LIN {X 0,Y 229.737,Z 261.729,A -85,B 0,C 180,E1 -19927.308,E2 -19927.308} C_VEL
LIN {X 0,Y 228.307,Z 255.768,A -85,B 0,C 180,E1 -19931.044,E2 -19931.044} C_VEL
LIN {X 0,Y 227.847,Z 253.604,A -85,B 0,C 180,E1 -19932.574,E2 -19932.574} C_VEL
LIN {X 0,Y 227.809,Z 253.608,A -85,B 0,C 180,E1 -19937.256,E2 -19937.256} C_VEL
LIN {X 0,Y 227.847,Z 253.599,A -85,B 0,C 180,E1 -19941.908,E2 -19941.908} C_VEL
LIN {X 0,Y 227.882,Z 253.572,A -85,B 0,C 180,E1 -19946.376,E2 -19946.376} C_VEL
LIN {X 0,Y 227.906,Z 253.589,A -85,B 0,C 180,E1 -19950.435,E2 -19950.435} C_VEL
LIN {X 0,Y 227.93,Z 253.565,A -85,B 0,C 180,E1 -19954.425,E2 -19954.425} C_VEL
LIN {X 0,Y 227.963,Z 253.579,A -85,B 0,C 180,E1 -19958.286,E2 -19958.286} C_VEL
LIN {X 0,Y 228.005,Z 253.549,A -85,B 0,C 180,E1 -19962.85,E2 -19962.85} C_VEL
LIN {X 0,Y 228.067,Z 253.561,A -85,B 0,C 180,E1 -19967.542,E2 -19967.542} C_VEL
LIN {X 0,Y 228.255,Z 253.506,A -85,B 0,C 180,E1 -19971.143,E2 -19971.143} C_VEL
LIN {X 0,Y 228.306,Z 253.525,A -85,B 0,C 180,E1 -19972.926,E2 -19972.926} C_VEL
LIN {X 0,Y 228.553,Z 253.484,A -85,B 0,C 180,E1 -19978.237,E2 -19978.237} C_VEL
LIN {X 0,Y 228.554,Z 253.477,A -85,B 0,C 180,E1 -19981.761,E2 -19981.761} C_VEL
LIN {X 0,Y 228.339,Z 253.528,A -85,B 0,C 180,E1 -19987.071,E2 -19987.071} C_VEL
LIN {X 0,Y 228.145,Z 253.521,A -85,B 0,C 180,E1 -19990.65,E2 -19990.65} C_VEL
LIN {X 0,Y 228.064,Z 253.576,A -85,B 0,C 180,E1 -19994.271,E2 -19994.271} C_VEL
LIN {X 0,Y 228.001,Z 253.548,A -85,B 0,C 180,E1 -19997.952,E2 -19997.952} C_VEL
LIN {X 0,Y 227.915,Z 253.589,A -85,B 0,C 180,E1 -20002.32,E2 -20002.32} C_VEL
LIN {X 0,Y 227.939,Z 253.559,A -85,B 0,C 180,E1 -20006.601,E2 -20006.601} C_VEL
LIN {X 0,Y 227.895,Z 253.595,A -85,B 0,C 180,E1 -20010.29,E2 -20010.29} C_VEL
LIN {X 0,Y 227.887,Z 253.575,A -85,B 0,C 180,E1 -20013.717,E2 -20013.717} C_VEL
LIN {X 0,Y 227.869,Z 253.602,A -85,B 0,C 180,E1 -20018.085,E2 -20018.085} C_VEL
LIN {X 0,Y 227.907,Z 253.592,A -85,B 0,C 180,E1 -20022.719,E2 -20022.719} C_VEL
LIN {X 0,Y 227.818,Z 253.543,A -85,B 0,C 180,E1 -20027.259,E2 -20027.259} C_VEL
LIN {X 0,Y 227.867,Z 253.603,A -85,B 0,C 180,E1 -20031.914,E2 -20031.914} C_VEL
LIN {X 0,Y 227.936,Z 253.841,A -85,B 0,C 180,E1 -20032.886,E2 -20032.886} C_VEL
LIN {X 0,Y 228.192,Z 254.913,A -85,B 0,C 180,E1 -20033.201,E2 -20033.201} C_VEL
LIN {X 0,Y 229.812,Z 257.623,A -85,B 0,C 180,E1 -20033.627,E2 -20033.627} C_VEL
LIN {X 0,Y 237.856,Z 271.226,A -85,B 0,C 180,E1 -20035.542,E2 -20035.542} C_VEL
LIN {X 0,Y 245.107,Z 285.042,A -85,B 0,C 180,E1 -20037.18,E2 -20037.18} C_VEL
LIN {X 0,Y 252.288,Z 298.523,A -85,B 0,C 180,E1 -20038.675,E2 -20038.675} C_VEL
LIN {X 0,Y 261.001,Z 311.411,A -85,B 0,C 180,E1 -20040.242,E2 -20040.242} C_VEL
LIN {X 0,Y 271.599,Z 324.085,A -85,B 0,C 180,E1 -20041.896,E2 -20041.896} C_VEL
LIN {X 0,Y 286.219,Z 338.842,A -85,B 0,C 180,E1 -20043.865,E2 -20043.865} C_VEL
LIN {X 0,Y 299.817,Z 350.422,A -85,B 0,C 180,E1 -20045.476,E2 -20045.476} C_VEL
LIN {X 0,Y 307.35,Z 356.574,A -85,B 0,C 180,E1 -20046.45,E2 -20046.45} C_VEL
LIN {X 0,Y 315.79,Z 363.116,A -85,B 0,C 180,E1 -20047.769,E2 -20047.769} C_VEL
LIN {X 0,Y 323.958,Z 369.179,A -85,B 0,C 180,E1 -20049.245,E2 -20049.245} C_VEL
LIN {X 0,Y 332.274,Z 375.418,A -85,B 0,C 180,E1 -20050.97,E2 -20050.97} C_VEL
LIN {X 0,Y 339.722,Z 380.424,A -85,B 0,C 180,E1 -20052.688,E2 -20052.688} C_VEL
LIN {X 0,Y 346.418,Z 385.336,A -85,B 0,C 180,E1 -20054.487,E2 -20054.487} C_VEL
LIN {X 0,Y 351.921,Z 388.859,A -85,B 0,C 180,E1 -20056.134,E2 -20056.134} C_VEL
LIN {X 0,Y 355.938,Z 391.12,A -85,B 0,C 180,E1 -20057.456,E2 -20057.456} C_VEL
LIN {X 0,Y 359.128,Z 393.588,A -85,B 0,C 180,E1 -20058.715,E2 -20058.715} C_VEL
LIN {X 0,Y 363.313,Z 396.472,A -85,B 0,C 180,E1 -20060.589,E2 -20060.589} C_VEL
LIN {X 0,Y 366.571,Z 398.29,A -85,B 0,C 180,E1 -20062.287,E2 -20062.287} C_VEL
LIN {X 0,Y 368.408,Z 399.219,A -85,B 0,C 180,E1 -20063.428,E2 -20063.428} C_VEL
LIN {X 0,Y 369.965,Z 399.891,A -85,B 0,C 180,E1 -20064.55,E2 -20064.55} C_VEL
LIN {X 0,Y 371.247,Z 400.329,A -85,B 0,C 180,E1 -20065.657,E2 -20065.657} C_VEL
LIN {X 0,Y 372.236,Z 400.623,A -85,B 0,C 180,E1 -20066.753,E2 -20066.753} C_VEL
LIN {X 0,Y 372.866,Z 401.006,A -85,B 0,C 180,E1 -20067.84,E2 -20067.84} C_VEL
LIN {X 0,Y 373.231,Z 401.261,A -85,B 0,C 180,E1 -20068.921,E2 -20068.921} C_VEL
LIN {X 0,Y 373.406,Z 401.192,A -85,B 0,C 180,E1 -20070,E2 -20070} C_VEL
LIN {X 0,Y 373.242,Z 401.224,A -85,B 0,C 180,E1 -20071.079,E2 -20071.079} C_VEL
LIN {X 0,Y 372.799,Z 400.889,A -85,B 0,C 180,E1 -20072.374,E2 -20072.374} C_VEL
LIN {X 0,Y 371.247,Z 400.335,A -85,B 0,C 180,E1 -20074.343,E2 -20074.343} C_VEL
LIN {X 0,Y 369.963,Z 399.917,A -85,B 0,C 180,E1 -20075.45,E2 -20075.45} C_VEL
LIN {X 0,Y 368.056,Z 399.053,A -85,B 0,C 180,E1 -20076.821,E2 -20076.821} C_VEL
LIN {X 0,Y 364.414,Z 397.149,A -85,B 0,C 180,E1 -20078.875,E2 -20078.875} C_VEL
LIN {X 0,Y 361.943,Z 395.593,A -85,B 0,C 180,E1 -20080.064,E2 -20080.064} C_VEL
LIN {X 0,Y 357.635,Z 392.463,A -85,B 0,C 180,E1 -20081.885,E2 -20081.885} C_VEL
LIN {X 0,Y 355.91,Z 391.059,A -85,B 0,C 180,E1 -20082.545,E2 -20082.545} C_VEL
LIN {X 0,Y 351.917,Z 388.848,A -85,B 0,C 180,E1 -20083.866,E2 -20083.866} C_VEL
LIN {X 0,Y 345.895,Z 385.025,A -85,B 0,C 180,E1 -20085.654,E2 -20085.654} C_VEL
LIN {X 0,Y 339.248,Z 380.069,A -85,B 0,C 180,E1 -20087.431,E2 -20087.431} C_VEL
LIN {X 0,Y 331.554,Z 374.906,A -85,B 0,C 180,E1 -20089.184,E2 -20089.184} C_VEL
LIN {X 0,Y 323.397,Z 368.785,A -85,B 0,C 180,E1 -20090.86,E2 -20090.86} C_VEL
LIN {X 0,Y 315.566,Z 362.953,A -85,B 0,C 180,E1 -20092.266,E2 -20092.266} C_VEL
LIN {X 0,Y 307.371,Z 356.596,A -85,B 0,C 180,E1 -20093.548,E2 -20093.548} C_VEL
LIN {X 0,Y 299.818,Z 350.408,A -85,B 0,C 180,E1 -20094.525,E2 -20094.525} C_VEL
LIN {X 0,Y 286.642,Z 339.218,A -85,B 0,C 180,E1 -20096.082,E2 -20096.082} C_VEL
LIN {X 0,Y 271.943,Z 324.45,A -85,B 0,C 180,E1 -20098.055,E2 -20098.055} C_VEL
LIN {X 0,Y 261.435,Z 311.99,A -85,B 0,C 180,E1 -20099.685,E2 -20099.685} C_VEL
LIN {X 0,Y 252.682,Z 299.196,A -85,B 0,C 180,E1 -20101.248,E2 -20101.248} C_VEL
LIN {X 0,Y 245.461,Z 285.814,A -85,B 0,C 180,E1 -20102.74,E2 -20102.74} C_VEL
LIN {X 0,Y 239.261,Z 273.837,A -85,B 0,C 180,E1 -20104.133,E2 -20104.133} C_VEL
LIN {X 0,Y 231.483,Z 260.425,A -85,B 0,C 180,E1 -20105.961,E2 -20105.961} C_VEL
LIN {X 0,Y 229.703,Z 257.505,A -85,B 0,C 180,E1 -20106.397,E2 -20106.397} C_VEL
LIN {X 0,Y 228.093,Z 254.532,A -85,B 0,C 180,E1 -20106.86,E2 -20106.86} C_VEL
LIN {X 0,Y 227.902,Z 253.655,A -85,B 0,C 180,E1 -20107.312,E2 -20107.312} C_VEL
LIN {X 0,Y 227.832,Z 253.551,A -85,B 0,C 180,E1 -20110.375,E2 -20110.375} C_VEL
LIN {X 0,Y 227.854,Z 253.579,A -85,B 0,C 180,E1 -20115.187,E2 -20115.187} C_VEL
LIN {X 0,Y 227.907,Z 253.585,A -85,B 0,C 180,E1 -20117.739,E2 -20117.739} C_VEL
LIN {X 0,Y 227.869,Z 253.602,A -85,B 0,C 180,E1 -20121.915,E2 -20121.915} C_VEL
LIN {X 0,Y 227.888,Z 253.575,A -85,B 0,C 180,E1 -20126.374,E2 -20126.374} C_VEL
LIN {X 0,Y 227.902,Z 253.583,A -85,B 0,C 180,E1 -20130.437,E2 -20130.437} C_VEL
LIN {X 0,Y 227.923,Z 253.572,A -85,B 0,C 180,E1 -20134.426,E2 -20134.426} C_VEL
LIN {X 0,Y 227.946,Z 253.577,A -85,B 0,C 180,E1 -20138.287,E2 -20138.287} C_VEL
LIN {X 0,Y 228.033,Z 253.555,A -85,B 0,C 180,E1 -20142.827,E2 -20142.827} C_VEL
LIN {X 0,Y 228.072,Z 253.556,A -85,B 0,C 180,E1 -20147.544,E2 -20147.544} C_VEL
LIN {X 0,Y 228.267,Z 253.509,A -85,B 0,C 180,E1 -20151.146,E2 -20151.146} C_VEL
LIN {X 0,Y 228.339,Z 253.528,A -85,B 0,C 180,E1 -20152.929,E2 -20152.929} C_VEL
LIN {X 0,Y 228.554,Z 253.477,A -85,B 0,C 180,E1 -20158.239,E2 -20158.239} C_VEL
LIN {X 0,Y 228.553,Z 253.484,A -85,B 0,C 180,E1 -20161.763,E2 -20161.763} C_VEL
LIN {X 0,Y 228.306,Z 253.525,A -85,B 0,C 180,E1 -20167.074,E2 -20167.074} C_VEL
LIN {X 0,Y 228.145,Z 253.523,A -85,B 0,C 180,E1 -20170.652,E2 -20170.652} C_VEL
LIN {X 0,Y 228.046,Z 253.575,A -85,B 0,C 180,E1 -20174.274,E2 -20174.274} C_VEL
LIN {X 0,Y 227.971,Z 253.546,A -85,B 0,C 180,E1 -20177.957,E2 -20177.957} C_VEL
LIN {X 0,Y 227.931,Z 253.589,A -85,B 0,C 180,E1 -20182.33,E2 -20182.33} C_VEL
LIN {X 0,Y 227.943,Z 253.556,A -85,B 0,C 180,E1 -20186.603,E2 -20186.603} C_VEL
LIN {X 0,Y 227.898,Z 253.596,A -85,B 0,C 180,E1 -20190.292,E2 -20190.292} C_VEL
LIN {X 0,Y 227.88,Z 253.572,A -85,B 0,C 180,E1 -20193.721,E2 -20193.721} C_VEL
LIN {X 0,Y 227.847,Z 253.599,A -85,B 0,C 180,E1 -20198.092,E2 -20198.092} C_VEL
LIN {X 0,Y 227.809,Z 253.608,A -85,B 0,C 180,E1 -20202.744,E2 -20202.744} C_VEL
LIN {X 0,Y 227.847,Z 253.614,A -85,B 0,C 180,E1 -20207.426,E2 -20207.426} C_VEL
LIN {X 0,Y 229.235,Z 259.354,A -85,B 0,C 180,E1 -20211.232,E2 -20211.232} C_VEL
LIN {X 0,Y 230.078,Z 263.105,A -85,B 0,C 180,E1 -20213.398,E2 -20213.398} C_VEL
LIN {X 0,Y 231.753,Z 266.915,A -85,B 0,C 180,E1 -20213.949,E2 -20213.949} C_VEL
LIN {X 0,Y 238.319,Z 280.506,A -85,B 0,C 180,E1 -20215.569,E2 -20215.569} C_VEL
LIN {X 0,Y 243.678,Z 293.124,A -85,B 0,C 180,E1 -20216.858,E2 -20216.858} C_VEL
LIN {X 0,Y 247.512,Z 314.657,A -85,B 0,C 180,E1 -20218.153,E2 -20218.153} C_VEL
LIN {X 0,Y 248.126,Z 318.744,A -85,B 0,C 180,E1 -20218.376,E2 -20218.376} C_VEL
LIN {X 0,Y 248.041,Z 322.266,A -85,B 0,C 180,E1 -20218.481,E2 -20218.481} C_VEL
LIN {X 0,Y 247.222,Z 328.114,A -85,B 0,C 180,E1 -20218.56,E2 -20218.56} C_VEL
LIN {X 0,Y 241.565,Z 347.124,A -85,B 0,C 180,E1 -20218.394,E2 -20218.394} C_VEL
LIN {X 0,Y 240.803,Z 352.968,A -85,B 0,C 180,E1 -20218.483,E2 -20218.483} C_VEL
LIN {X 0,Y 239.893,Z 372.687,A -85,B 0,C 180,E1 -20219.125,E2 -20219.125} C_VEL
LIN {X 0,Y 238.345,Z 386.631,A -85,B 0,C 180,E1 -20219.916,E2 -20219.916} C_VEL
LIN {X 0,Y 236.753,Z 397.271,A -85,B 0,C 180,E1 -20220.795,E2 -20220.795} C_VEL
LIN {X 0,Y 235.174,Z 405.775,A -85,B 0,C 180,E1 -20221.679,E2 -20221.679} C_VEL
LIN {X 0,Y 233.292,Z 415.049,A -85,B 0,C 180,E1 -20222.894,E2 -20222.894} C_VEL
LIN {X 0,Y 231.234,Z 423.992,A -85,B 0,C 180,E1 -20224.335,E2 -20224.335} C_VEL
LIN {X 0,Y 228.992,Z 432.516,A -85,B 0,C 180,E1 -20226.005,E2 -20226.005} C_VEL
LIN {X 0,Y 227.037,Z 439.733,A -85,B 0,C 180,E1 -20227.716,E2 -20227.716} C_VEL
LIN {X 0,Y 225.477,Z 445.825,A -85,B 0,C 180,E1 -20229.433,E2 -20229.433} C_VEL
LIN {X 0,Y 223.485,Z 452.473,A -85,B 0,C 180,E1 -20231.671,E2 -20231.671} C_VEL
LIN {X 0,Y 222.243,Z 456.976,A -85,B 0,C 180,E1 -20233.465,E2 -20233.465} C_VEL
LIN {X 0,Y 220.61,Z 462.466,A -85,B 0,C 180,E1 -20236.177,E2 -20236.177} C_VEL
LIN {X 0,Y 219.587,Z 466.796,A -85,B 0,C 180,E1 -20238.929,E2 -20238.929} C_VEL
LIN {X 0,Y 219.086,Z 469.166,A -85,B 0,C 180,E1 -20240.77,E2 -20240.77} C_VEL
LIN {X 0,Y 218.737,Z 470.968,A -85,B 0,C 180,E1 -20242.616,E2 -20242.616} C_VEL
LIN {X 0,Y 218.501,Z 473.423,A -85,B 0,C 180,E1 -20246.312,E2 -20246.312} C_VEL
LIN {X 0,Y 218.524,Z 474.016,A -85,B 0,C 180,E1 -20248.157,E2 -20248.157} C_VEL
LIN {X 0,Y 218.623,Z 474.174,A -85,B 0,C 180,E1 -20250,E2 -20250} C_VEL
LIN {X 0,Y 218.524,Z 474.016,A -85,B 0,C 180,E1 -20251.843,E2 -20251.843} C_VEL
LIN {X 0,Y 218.484,Z 473.159,A -85,B 0,C 180,E1 -20254.292,E2 -20254.292} C_VEL
LIN {X 0,Y 218.705,Z 470.967,A -85,B 0,C 180,E1 -20257.385,E2 -20257.385} C_VEL
LIN {X 0,Y 219.314,Z 468.015,A -85,B 0,C 180,E1 -20260.151,E2 -20260.151} C_VEL
LIN {X 0,Y 220.223,Z 464.022,A -85,B 0,C 180,E1 -20262.908,E2 -20262.908} C_VEL
LIN {X 0,Y 221.649,Z 458.891,A -85,B 0,C 180,E1 -20265.635,E2 -20265.635} C_VEL
LIN {X 0,Y 223.148,Z 453.628,A -85,B 0,C 180,E1 -20267.883,E2 -20267.883} C_VEL
LIN {X 0,Y 225.05,Z 447.314,A -85,B 0,C 180,E1 -20270.091,E2 -20270.091} C_VEL
LIN {X 0,Y 226.622,Z 441.361,A -85,B 0,C 180,E1 -20271.848,E2 -20271.848} C_VEL
LIN {X 0,Y 228.482,Z 434.435,A -85,B 0,C 180,E1 -20273.57,E2 -20273.57} C_VEL
LIN {X 0,Y 230.686,Z 426.261,A -85,B 0,C 180,E1 -20275.247,E2 -20275.247} C_VEL
LIN {X 0,Y 232.7,Z 417.752,A -85,B 0,C 180,E1 -20276.696,E2 -20276.696} C_VEL
LIN {X 0,Y 234.562,Z 409.039,A -85,B 0,C 180,E1 -20277.915,E2 -20277.915} C_VEL
LIN {X 0,Y 236.239,Z 400.291,A -85,B 0,C 180,E1 -20278.91,E2 -20278.91} C_VEL
LIN {X 0,Y 237.837,Z 390.494,A -85,B 0,C 180,E1 -20279.789,E2 -20279.789} C_VEL
LIN {X 0,Y 239.069,Z 380.72,A -85,B 0,C 180,E1 -20280.46,E2 -20280.46} C_VEL
LIN {X 0,Y 240.014,Z 370.366,A -85,B 0,C 180,E1 -20280.964,E2 -20280.964} C_VEL
LIN {X 0,Y 241.204,Z 343.742,A -85,B 0,C 180,E1 -20281.774,E2 -20281.774} C_VEL
LIN {X 0,Y 241.982,Z 319.229,A -85,B 0,C 180,E1 -20282.501,E2 -20282.501} C_VEL
LIN {X 0,Y 238.66,Z 299.408,A -85,B 0,C 180,E1 -20283.704,E2 -20283.704} C_VEL
LIN {X 0,Y 237.524,Z 294.652,A -85,B 0,C 180,E1 -20284.056,E2 -20284.056} C_VEL
LIN {X 0,Y 230.872,Z 279.383,A -85,B 0,C 180,E1 -20285.74,E2 -20285.74} C_VEL
LIN {X 0,Y 224.408,Z 266.483,A -85,B 0,C 180,E1 -20287.435,E2 -20287.435} C_VEL
LIN {X 0,Y 222.795,Z 262.883,A -85,B 0,C 180,E1 -20287.999,E2 -20287.999} C_VEL
LIN {X 0,Y 221.307,Z 256.828,A -85,B 0,C 180,E1 -20291.827,E2 -20291.827} C_VEL
LIN {X 0,Y 220.77,Z 254.494,A -85,B 0,C 180,E1 -20293.614,E2 -20293.614} C_VEL
LIN {X 0,Y 220.769,Z 254.482,A -85,B 0,C 180,E1 -20298.046,E2 -20298.046} C_VEL
LIN {X 0,Y 220.826,Z 254.479,A -85,B 0,C 180,E1 -20302.792,E2 -20302.792} C_VEL
LIN {X 0,Y 220.818,Z 254.458,A -85,B 0,C 180,E1 -20307.243,E2 -20307.243} C_VEL
LIN {X 0,Y 220.828,Z 254.453,A -85,B 0,C 180,E1 -20311.484,E2 -20311.484} C_VEL
LIN {X 0,Y 220.869,Z 254.459,A -85,B 0,C 180,E1 -20315.564,E2 -20315.564} C_VEL
LIN {X 0,Y 220.889,Z 254.44,A -85,B 0,C 180,E1 -20319.513,E2 -20319.513} C_VEL
LIN {X 0,Y 220.987,Z 254.43,A -85,B 0,C 180,E1 -20323.367,E2 -20323.367} C_VEL
LIN {X 0,Y 221.004,Z 254.445,A -85,B 0,C 180,E1 -20327.137,E2 -20327.137} C_VEL
LIN {X 0,Y 221.195,Z 254.383,A -85,B 0,C 180,E1 -20330.858,E2 -20330.858} C_VEL
LIN {X 0,Y 221.129,Z 254.437,A -85,B 0,C 180,E1 -20334.528,E2 -20334.528} C_VEL
LIN {X 0,Y 221.511,Z 254.361,A -85,B 0,C 180,E1 -20338.181,E2 -20338.181} C_VEL
LIN {X 0,Y 221.512,Z 254.353,A -85,B 0,C 180,E1 -20341.817,E2 -20341.817} C_VEL
LIN {X 0,Y 221.271,Z 254.402,A -85,B 0,C 180,E1 -20347.298,E2 -20347.298} C_VEL
LIN {X 0,Y 221.067,Z 254.405,A -85,B 0,C 180,E1 -20350.995,E2 -20350.995} C_VEL
LIN {X 0,Y 220.996,Z 254.458,A -85,B 0,C 180,E1 -20354.738,E2 -20354.738} C_VEL
LIN {X 0,Y 220.919,Z 254.425,A -85,B 0,C 180,E1 -20358.549,E2 -20358.549} C_VEL
LIN {X 0,Y 220.883,Z 254.468,A -85,B 0,C 180,E1 -20362.675,E2 -20362.675} C_VEL
LIN {X 0,Y 220.881,Z 254.436,A -85,B 0,C 180,E1 -20367.013,E2 -20367.013} C_VEL
LIN {X 0,Y 220.836,Z 254.479,A -85,B 0,C 180,E1 -20370.767,E2 -20370.767} C_VEL
LIN {X 0,Y 220.813,Z 254.453,A -85,B 0,C 180,E1 -20374.951,E2 -20374.951} C_VEL
LIN {X 0,Y 220.853,Z 254.458,A -85,B 0,C 180,E1 -20379.525,E2 -20379.525} C_VEL
LIN {X 0,Y 220.864,Z 254.472,A -85,B 0,C 180,E1 -20382.957,E2 -20382.957} C_VEL
LIN {X 0,Y 220.776,Z 254.417,A -85,B 0,C 180,E1 -20388.049,E2 -20388.049} C_VEL
LIN {X 0,Y 220.836,Z 254.701,A -85,B 0,C 180,E1 -20391.491,E2 -20391.491} C_VEL
LIN {X 0,Y 221.128,Z 255.823,A -85,B 0,C 180,E1 -20391.848,E2 -20391.848} C_VEL
LIN {X 0,Y 222.822,Z 258.61,A -85,B 0,C 180,E1 -20392.322,E2 -20392.322} C_VEL
LIN {X 0,Y 228.235,Z 267.33,A -85,B 0,C 180,E1 -20393.706,E2 -20393.706} C_VEL
LIN {X 0,Y 237.078,Z 283.229,A -85,B 0,C 180,E1 -20395.845,E2 -20395.845} C_VEL
LIN {X 0,Y 246.332,Z 301.326,A -85,B 0,C 180,E1 -20397.916,E2 -20397.916} C_VEL
LIN {X 0,Y 254.709,Z 314.108,A -85,B 0,C 180,E1 -20399.51,E2 -20399.51} C_VEL
LIN {X 0,Y 263.082,Z 324.749,A -85,B 0,C 180,E1 -20400.913,E2 -20400.913} C_VEL
LIN {X 0,Y 275.601,Z 338.122,A -85,B 0,C 180,E1 -20402.747,E2 -20402.747} C_VEL
LIN {X 0,Y 285.746,Z 347.624,A -85,B 0,C 180,E1 -20404.06,E2 -20404.06} C_VEL
LIN {X 0,Y 296.508,Z 356.709,A -85,B 0,C 180,E1 -20405.344,E2 -20405.344} C_VEL
LIN {X 0,Y 304.924,Z 363.572,A -85,B 0,C 180,E1 -20406.474,E2 -20406.474} C_VEL
LIN {X 0,Y 312.969,Z 369.81,A -85,B 0,C 180,E1 -20407.749,E2 -20407.749} C_VEL
LIN {X 0,Y 321.3,Z 375.892,A -85,B 0,C 180,E1 -20409.254,E2 -20409.254} C_VEL
LIN {X 0,Y 329.279,Z 381.914,A -85,B 0,C 180,E1 -20410.917,E2 -20410.917} C_VEL
LIN {X 0,Y 335.925,Z 386.279,A -85,B 0,C 180,E1 -20412.433,E2 -20412.433} C_VEL
LIN {X 0,Y 343.054,Z 391.525,A -85,B 0,C 180,E1 -20414.334,E2 -20414.334} C_VEL
LIN {X 0,Y 348.695,Z 395.135,A -85,B 0,C 180,E1 -20416.004,E2 -20416.004} C_VEL
LIN {X 0,Y 352.899,Z 397.518,A -85,B 0,C 180,E1 -20417.376,E2 -20417.376} C_VEL
LIN {X 0,Y 357.622,Z 401.061,A -85,B 0,C 180,E1 -20419.292,E2 -20419.292} C_VEL
LIN {X 0,Y 361.371,Z 403.495,A -85,B 0,C 180,E1 -20421.049,E2 -20421.049} C_VEL
LIN {X 0,Y 363.553,Z 404.71,A -85,B 0,C 180,E1 -20422.223,E2 -20422.223} C_VEL
LIN {X 0,Y 365.44,Z 405.641,A -85,B 0,C 180,E1 -20423.374,E2 -20423.374} C_VEL
LIN {X 0,Y 367.1,Z 406.372,A -85,B 0,C 180,E1 -20424.567,E2 -20424.567} C_VEL
LIN {X 0,Y 368.316,Z 406.802,A -85,B 0,C 180,E1 -20425.623,E2 -20425.623} C_VEL
LIN {X 0,Y 369.338,Z 407.082,A -85,B 0,C 180,E1 -20426.727,E2 -20426.727} C_VEL
LIN {X 0,Y 369.973,Z 407.466,A -85,B 0,C 180,E1 -20427.823,E2 -20427.823} C_VEL
LIN {X 0,Y 370.328,Z 407.739,A -85,B 0,C 180,E1 -20428.913,E2 -20428.913} C_VEL
LIN {X 0,Y 370.524,Z 407.653,A -85,B 0,C 180,E1 -20430,E2 -20430} C_VEL
LIN {X 0,Y 370.339,Z 407.699,A -85,B 0,C 180,E1 -20431.087,E2 -20431.087} C_VEL
LIN {X 0,Y 369.982,Z 407.421,A -85,B 0,C 180,E1 -20432.177,E2 -20432.177} C_VEL
LIN {X 0,Y 369.321,Z 407.091,A -85,B 0,C 180,E1 -20433.273,E2 -20433.273} C_VEL
LIN {X 0,Y 368.309,Z 406.791,A -85,B 0,C 180,E1 -20434.377,E2 -20434.377} C_VEL
LIN {X 0,Y 366.999,Z 406.368,A -85,B 0,C 180,E1 -20435.494,E2 -20435.494} C_VEL
LIN {X 0,Y 365.437,Z 405.653,A -85,B 0,C 180,E1 -20436.626,E2 -20436.626} C_VEL
LIN {X 0,Y 362.34,Z 404.069,A -85,B 0,C 180,E1 -20438.433,E2 -20438.433} C_VEL
LIN {X 0,Y 358.848,Z 401.956,A -85,B 0,C 180,E1 -20440.152,E2 -20440.152} C_VEL
LIN {X 0,Y 354.944,Z 399.137,A -85,B 0,C 180,E1 -20441.817,E2 -20441.817} C_VEL
LIN {X 0,Y 352.819,Z 397.42,A -85,B 0,C 180,E1 -20442.657,E2 -20442.657} C_VEL
LIN {X 0,Y 347.992,Z 394.719,A -85,B 0,C 180,E1 -20444.213,E2 -20444.213} C_VEL
LIN {X 0,Y 343.049,Z 391.521,A -85,B 0,C 180,E1 -20445.663,E2 -20445.663} C_VEL
LIN {X 0,Y 338.091,Z 387.913,A -85,B 0,C 180,E1 -20447.02,E2 -20447.02} C_VEL
LIN {X 0,Y 330.721,Z 382.898,A -85,B 0,C 180,E1 -20448.764,E2 -20448.764} C_VEL
LIN {X 0,Y 323.265,Z 377.334,A -85,B 0,C 180,E1 -20450.356,E2 -20450.356} C_VEL
LIN {X 0,Y 314.816,Z 371.22,A -85,B 0,C 180,E1 -20451.933,E2 -20451.933} C_VEL
LIN {X 0,Y 306.561,Z 364.81,A -85,B 0,C 180,E1 -20453.282,E2 -20453.282} C_VEL
LIN {X 0,Y 298.556,Z 358.454,A -85,B 0,C 180,E1 -20454.4,E2 -20454.4} C_VEL
LIN {X 0,Y 286.312,Z 348.104,A -85,B 0,C 180,E1 -20455.872,E2 -20455.872} C_VEL
LIN {X 0,Y 277.23,Z 339.708,A -85,B 0,C 180,E1 -20457.033,E2 -20457.033} C_VEL
LIN {X 0,Y 264.731,Z 326.645,A -85,B 0,C 180,E1 -20458.83,E2 -20458.83} C_VEL
LIN {X 0,Y 255.685,Z 315.463,A -85,B 0,C 180,E1 -20460.317,E2 -20460.317} C_VEL
LIN {X 0,Y 247.025,Z 302.541,A -85,B 0,C 180,E1 -20461.941,E2 -20461.941} C_VEL
LIN {X 0,Y 239.834,Z 288.77,A -85,B 0,C 180,E1 -20463.511,E2 -20463.511} C_VEL
LIN {X 0,Y 233.735,Z 277.07,A -85,B 0,C 180,E1 -20464.944,E2 -20464.944} C_VEL
LIN {X 0,Y 225.478,Z 262.702,A -85,B 0,C 180,E1 -20466.995,E2 -20466.995} C_VEL
LIN {X 0,Y 222.504,Z 258.225,A -85,B 0,C 180,E1 -20467.757,E2 -20467.757} C_VEL
LIN {X 0,Y 221.011,Z 255.468,A -85,B 0,C 180,E1 -20468.213,E2 -20468.213} C_VEL
LIN {X 0,Y 220.832,Z 254.537,A -85,B 0,C 180,E1 -20468.676,E2 -20468.676} C_VEL
LIN {X 0,Y 220.772,Z 254.421,A -85,B 0,C 180,E1 -20472.933,E2 -20472.933} C_VEL
LIN {X 0,Y 220.864,Z 254.472,A -85,B 0,C 180,E1 -20477.043,E2 -20477.043} C_VEL
LIN {X 0,Y 220.853,Z 254.458,A -85,B 0,C 180,E1 -20480.475,E2 -20480.475} C_VEL
LIN {X 0,Y 220.813,Z 254.453,A -85,B 0,C 180,E1 -20485.049,E2 -20485.049} C_VEL
LIN {X 0,Y 220.832,Z 254.477,A -85,B 0,C 180,E1 -20489.391,E2 -20489.391} C_VEL
LIN {X 0,Y 220.892,Z 254.437,A -85,B 0,C 180,E1 -20493.55,E2 -20493.55} C_VEL
LIN {X 0,Y 220.864,Z 254.469,A -85,B 0,C 180,E1 -20497.553,E2 -20497.553} C_VEL
LIN {X 0,Y 220.983,Z 254.428,A -85,B 0,C 180,E1 -20502.572,E2 -20502.572} C_VEL
LIN {X 0,Y 221.011,Z 254.441,A -85,B 0,C 180,E1 -20507.14,E2 -20507.14} C_VEL
LIN {X 0,Y 221.204,Z 254.386,A -85,B 0,C 180,E1 -20510.86,E2 -20510.86} C_VEL
LIN {X 0,Y 221.271,Z 254.402,A -85,B 0,C 180,E1 -20512.702,E2 -20512.702} C_VEL
LIN {X 0,Y 221.512,Z 254.353,A -85,B 0,C 180,E1 -20518.183,E2 -20518.183} C_VEL
LIN {X 0,Y 221.511,Z 254.361,A -85,B 0,C 180,E1 -20521.819,E2 -20521.819} C_VEL
LIN {X 0,Y 221.243,Z 254.398,A -85,B 0,C 180,E1 -20527.301,E2 -20527.301} C_VEL
LIN {X 0,Y 221.066,Z 254.407,A -85,B 0,C 180,E1 -20530.997,E2 -20530.997} C_VEL
LIN {X 0,Y 220.974,Z 254.455,A -85,B 0,C 180,E1 -20534.741,E2 -20534.741} C_VEL
LIN {X 0,Y 220.903,Z 254.424,A -85,B 0,C 180,E1 -20538.552,E2 -20538.552} C_VEL
LIN {X 0,Y 220.897,Z 254.467,A -85,B 0,C 180,E1 -20542.683,E2 -20542.683} C_VEL
LIN {X 0,Y 220.885,Z 254.434,A -85,B 0,C 180,E1 -20547.015,E2 -20547.015} C_VEL
LIN {X 0,Y 220.84,Z 254.477,A -85,B 0,C 180,E1 -20550.768,E2 -20550.768} C_VEL
LIN {X 0,Y 220.804,Z 254.455,A -85,B 0,C 180,E1 -20554.956,E2 -20554.956} C_VEL
LIN {X 0,Y 220.808,Z 254.462,A -85,B 0,C 180,E1 -20559.538,E2 -20559.538} C_VEL
LIN {X 0,Y 220.772,Z 254.472,A -85,B 0,C 180,E1 -20564.456,E2 -20564.456} C_VEL
LIN {X 0,Y 220.775,Z 254.624,A -85,B 0,C 180,E1 -20566.647,E2 -20566.647} C_VEL
LIN {X 0,Y 222.635,Z 262.158,A -85,B 0,C 180,E1 -20571.653,E2 -20571.653} C_VEL
LIN {X 0,Y 222.974,Z 263.405,A -85,B 0,C 180,E1 -20572.124,E2 -20572.124} C_VEL
LIN {X 0,Y 229.761,Z 277.101,A -85,B 0,C 180,E1 -20573.975,E2 -20573.975} C_VEL
LIN {X 0,Y 235.913,Z 290.708,A -85,B 0,C 180,E1 -20575.539,E2 -20575.539} C_VEL
LIN {X 0,Y 238.131,Z 296.44,A -85,B 0,C 180,E1 -20576.106,E2 -20576.106} C_VEL
LIN {X 0,Y 241.983,Z 319.204,A -85,B 0,C 180,E1 -20577.499,E2 -20577.499} C_VEL
LIN {X 0,Y 240.803,Z 352.968,A -85,B 0,C 180,E1 -20578.483,E2 -20578.483} C_VEL
LIN {X 0,Y 240.027,Z 358.812,A -85,B 0,C 180,E1 -20578.568,E2 -20578.568} C_VEL
LIN {X 0,Y 237.091,Z 368.287,A -85,B 0,C 180,E1 -20578.513,E2 -20578.513} C_VEL
LIN {X 0,Y 233.87,Z 377.68,A -85,B 0,C 180,E1 -20578.571,E2 -20578.571} C_VEL
LIN {X 0,Y 232.653,Z 383.395,A -85,B 0,C 180,E1 -20578.816,E2 -20578.816} C_VEL
LIN {X 0,Y 230.76,Z 396.072,A -85,B 0,C 180,E1 -20579.833,E2 -20579.833} C_VEL
LIN {X 0,Y 228.946,Z 405.582,A -85,B 0,C 180,E1 -20580.836,E2 -20580.836} C_VEL
LIN {X 0,Y 226.999,Z 414.857,A -85,B 0,C 180,E1 -20582.078,E2 -20582.078} C_VEL
LIN {X 0,Y 224.834,Z 423.799,A -85,B 0,C 180,E1 -20583.549,E2 -20583.549} C_VEL
LIN {X 0,Y 222.501,Z 432.323,A -85,B 0,C 180,E1 -20585.259,E2 -20585.259} C_VEL
LIN {X 0,Y 220.45,Z 439.54,A -85,B 0,C 180,E1 -20587.012,E2 -20587.012} C_VEL
LIN {X 0,Y 218.362,Z 447.121,A -85,B 0,C 180,E1 -20589.266,E2 -20589.266} C_VEL
LIN {X 0,Y 216.363,Z 453.435,A -85,B 0,C 180,E1 -20591.536,E2 -20591.536} C_VEL
LIN {X 0,Y 214.781,Z 458.697,A -85,B 0,C 180,E1 -20593.851,E2 -20593.851} C_VEL
LIN {X 0,Y 213.258,Z 463.828,A -85,B 0,C 180,E1 -20596.663,E2 -20596.663} C_VEL
LIN {X 0,Y 212.301,Z 467.821,A -85,B 0,C 180,E1 -20599.51,E2 -20599.51} C_VEL
LIN {X 0,Y 211.671,Z 470.775,A -85,B 0,C 180,E1 -20602.368,E2 -20602.368} C_VEL
LIN {X 0,Y 211.4,Z 473.23,A -85,B 0,C 180,E1 -20606.188,E2 -20606.188} C_VEL
LIN {X 0,Y 211.427,Z 473.823,A -85,B 0,C 180,E1 -20608.095,E2 -20608.095} C_VEL
LIN {X 0,Y 211.539,Z 473.982,A -85,B 0,C 180,E1 -20610,E2 -20610} C_VEL
LIN {X 0,Y 211.426,Z 473.823,A -85,B 0,C 180,E1 -20611.905,E2 -20611.905} C_VEL
LIN {X 0,Y 211.396,Z 473.114,A -85,B 0,C 180,E1 -20614.145,E2 -20614.145} C_VEL
LIN {X 0,Y 211.646,Z 470.774,A -85,B 0,C 180,E1 -20617.633,E2 -20617.633} C_VEL
LIN {X 0,Y 212.301,Z 467.821,A -85,B 0,C 180,E1 -20620.49,E2 -20620.49} C_VEL
LIN {X 0,Y 213.258,Z 463.828,A -85,B 0,C 180,E1 -20623.337,E2 -20623.337} C_VEL
LIN {X 0,Y 214.78,Z 458.697,A -85,B 0,C 180,E1 -20626.149,E2 -20626.149} C_VEL
LIN {X 0,Y 216.356,Z 453.434,A -85,B 0,C 180,E1 -20628.464,E2 -20628.464} C_VEL
LIN {X 0,Y 218.364,Z 447.121,A -85,B 0,C 180,E1 -20630.734,E2 -20630.734} C_VEL
LIN {X 0,Y 220.012,Z 441.167,A -85,B 0,C 180,E1 -20632.54,E2 -20632.54} C_VEL
LIN {X 0,Y 221.989,Z 434.242,A -85,B 0,C 180,E1 -20634.303,E2 -20634.303} C_VEL
LIN {X 0,Y 224.271,Z 426.068,A -85,B 0,C 180,E1 -20636.022,E2 -20636.022} C_VEL
LIN {X 0,Y 226.378,Z 417.559,A -85,B 0,C 180,E1 -20637.503,E2 -20637.503} C_VEL
LIN {X 0,Y 228.306,Z 408.846,A -85,B 0,C 180,E1 -20638.75,E2 -20638.75} C_VEL
LIN {X 0,Y 230.054,Z 400.099,A -85,B 0,C 180,E1 -20639.764,E2 -20639.764} C_VEL
LIN {X 0,Y 231.69,Z 390.301,A -85,B 0,C 180,E1 -20640.663,E2 -20640.663} C_VEL
LIN {X 0,Y 233.049,Z 379.985,A -85,B 0,C 180,E1 -20641.374,E2 -20641.374} C_VEL
LIN {X 0,Y 234.009,Z 369.745,A -85,B 0,C 180,E1 -20641.87,E2 -20641.87} C_VEL
LIN {X 0,Y 235.51,Z 335.178,A -85,B 0,C 180,E1 -20642.934,E2 -20642.934} C_VEL
LIN {X 0,Y 235.971,Z 320.244,A -85,B 0,C 180,E1 -20643.392,E2 -20643.392} C_VEL
LIN {X 0,Y 232.647,Z 300.172,A -85,B 0,C 180,E1 -20644.663,E2 -20644.663} C_VEL
LIN {X 0,Y 231.683,Z 296.886,A -85,B 0,C 180,E1 -20644.948,E2 -20644.948} C_VEL
LIN {X 0,Y 225.441,Z 282.568,A -85,B 0,C 180,E1 -20646.609,E2 -20646.609} C_VEL
LIN {X 0,Y 219.357,Z 270.324,A -85,B 0,C 180,E1 -20648.288,E2 -20648.288} C_VEL
LIN {X 0,Y 216.806,Z 265.628,A -85,B 0,C 180,E1 -20649.014,E2 -20649.014} C_VEL
LIN {X 0,Y 215.424,Z 262.564,A -85,B 0,C 180,E1 -20649.574,E2 -20649.574} C_VEL
LIN {X 0,Y 213.771,Z 255.543,A -85,B 0,C 180,E1 -20654.351,E2 -20654.351} C_VEL
LIN {X 0,Y 213.718,Z 255.347,A -85,B 0,C 180,E1 -20659.142,E2 -20659.142} C_VEL
LIN {X 0,Y 213.746,Z 255.35,A -85,B 0,C 180,E1 -20663.711,E2 -20663.711} C_VEL
LIN {X 0,Y 213.769,Z 255.349,A -85,B 0,C 180,E1 -20668.262,E2 -20668.262} C_VEL
LIN {X 0,Y 213.828,Z 255.314,A -85,B 0,C 180,E1 -20672.602,E2 -20672.602} C_VEL
LIN {X 0,Y 213.854,Z 255.345,A -85,B 0,C 180,E1 -20676.952,E2 -20676.952} C_VEL
LIN {X 0,Y 213.918,Z 255.301,A -85,B 0,C 180,E1 -20682.8,E2 -20682.8} C_VEL
LIN {X 0,Y 213.943,Z 255.328,A -85,B 0,C 180,E1 -20686.705,E2 -20686.705} C_VEL
LIN {X 0,Y 214.135,Z 255.261,A -85,B 0,C 180,E1 -20690.554,E2 -20690.554} C_VEL
LIN {X 0,Y 214.09,Z 255.313,A -85,B 0,C 180,E1 -20694.347,E2 -20694.347} C_VEL
LIN {X 0,Y 214.444,Z 255.241,A -85,B 0,C 180,E1 -20698.121,E2 -20698.121} C_VEL
LIN {X 0,Y 214.546,Z 255.21,A -85,B 0,C 180,E1 -20699.999,E2 -20699.999} C_VEL
LIN {X 0,Y 214.445,Z 255.233,A -85,B 0,C 180,E1 -20701.877,E2 -20701.877} C_VEL
LIN {X 0,Y 214.208,Z 255.276,A -85,B 0,C 180,E1 -20707.54,E2 -20707.54} C_VEL
LIN {X 0,Y 213.999,Z 255.288,A -85,B 0,C 180,E1 -20711.363,E2 -20711.363} C_VEL
LIN {X 0,Y 213.934,Z 255.335,A -85,B 0,C 180,E1 -20715.236,E2 -20715.236} C_VEL
LIN {X 0,Y 213.834,Z 255.306,A -85,B 0,C 180,E1 -20719.187,E2 -20719.187} C_VEL
LIN {X 0,Y 213.809,Z 255.352,A -85,B 0,C 180,E1 -20723.23,E2 -20723.23} C_VEL
LIN {X 0,Y 213.827,Z 255.314,A -85,B 0,C 180,E1 -20727.449,E2 -20727.449} C_VEL
LIN {X 0,Y 213.768,Z 255.356,A -85,B 0,C 180,E1 -20731.736,E2 -20731.736} C_VEL
LIN {X 0,Y 213.753,Z 255.344,A -85,B 0,C 180,E1 -20736.285,E2 -20736.285} C_VEL
LIN {X 0,Y 213.791,Z 255.333,A -85,B 0,C 180,E1 -20741.105,E2 -20741.105} C_VEL
LIN {X 0,Y 213.806,Z 255.352,A -85,B 0,C 180,E1 -20743.684,E2 -20743.684} C_VEL
LIN {X 0,Y 213.716,Z 255.298,A -85,B 0,C 180,E1 -20748.876,E2 -20748.876} C_VEL
LIN {X 0,Y 213.831,Z 255.664,A -85,B 0,C 180,E1 -20750.083,E2 -20750.083} C_VEL
LIN {X 0,Y 214.247,Z 257.103,A -85,B 0,C 180,E1 -20750.442,E2 -20750.442} C_VEL
LIN {X 0,Y 215.915,Z 259.594,A -85,B 0,C 180,E1 -20750.924,E2 -20750.924} C_VEL
LIN {X 0,Y 223.419,Z 271.636,A -85,B 0,C 180,E1 -20752.958,E2 -20752.958} C_VEL
LIN {X 0,Y 231.868,Z 286.947,A -85,B 0,C 180,E1 -20755.098,E2 -20755.098} C_VEL
LIN {X 0,Y 241.222,Z 305.45,A -85,B 0,C 180,E1 -20757.29,E2 -20757.29} C_VEL
LIN {X 0,Y 249.147,Z 317.77,A -85,B 0,C 180,E1 -20758.869,E2 -20758.869} C_VEL
LIN {X 0,Y 257.001,Z 328.014,A -85,B 0,C 180,E1 -20760.253,E2 -20760.253} C_VEL
LIN {X 0,Y 269.628,Z 341.955,A -85,B 0,C 180,E1 -20762.199,E2 -20762.199} C_VEL
LIN {X 0,Y 281.297,Z 353.008,A -85,B 0,C 180,E1 -20763.776,E2 -20763.776} C_VEL
LIN {X 0,Y 291.892,Z 362.062,A -85,B 0,C 180,E1 -20765.148,E2 -20765.148} C_VEL
LIN {X 0,Y 301.776,Z 370.061,A -85,B 0,C 180,E1 -20766.499,E2 -20766.499} C_VEL
LIN {X 0,Y 308.378,Z 375.137,A -85,B 0,C 180,E1 -20767.533,E2 -20767.533} C_VEL
LIN {X 0,Y 316.304,Z 381.006,A -85,B 0,C 180,E1 -20768.937,E2 -20768.937} C_VEL
LIN {X 0,Y 323.614,Z 386.462,A -85,B 0,C 180,E1 -20770.408,E2 -20770.408} C_VEL
LIN {X 0,Y 330.78,Z 391.382,A -85,B 0,C 180,E1 -20772.005,E2 -20772.005} C_VEL
LIN {X 0,Y 337.829,Z 396.471,A -85,B 0,C 180,E1 -20773.814,E2 -20773.814} C_VEL
LIN {X 0,Y 341.976,Z 399.286,A -85,B 0,C 180,E1 -20774.992,E2 -20774.992} C_VEL
LIN {X 0,Y 346.923,Z 402.242,A -85,B 0,C 180,E1 -20776.501,E2 -20776.501} C_VEL
LIN {X 0,Y 350.595,Z 404.618,A -85,B 0,C 180,E1 -20777.783,E2 -20777.783} C_VEL
LIN {X 0,Y 355.23,Z 408.04,A -85,B 0,C 180,E1 -20779.743,E2 -20779.743} C_VEL
LIN {X 0,Y 357.785,Z 409.596,A -85,B 0,C 180,E1 -20780.959,E2 -20780.959} C_VEL
LIN {X 0,Y 361.225,Z 411.464,A -85,B 0,C 180,E1 -20782.859,E2 -20782.859} C_VEL
LIN {X 0,Y 363.571,Z 412.536,A -85,B 0,C 180,E1 -20784.454,E2 -20784.454} C_VEL
LIN {X 0,Y 364.921,Z 413.051,A -85,B 0,C 180,E1 -20785.582,E2 -20785.582} C_VEL
LIN {X 0,Y 366.043,Z 413.362,A -85,B 0,C 180,E1 -20786.741,E2 -20786.741} C_VEL
LIN {X 0,Y 366.654,Z 413.737,A -85,B 0,C 180,E1 -20787.803,E2 -20787.803} C_VEL
LIN {X 0,Y 367.011,Z 414.013,A -85,B 0,C 180,E1 -20788.903,E2 -20788.903} C_VEL
LIN {X 0,Y 367.232,Z 413.919,A -85,B 0,C 180,E1 -20790,E2 -20790} C_VEL
LIN {X 0,Y 367.027,Z 413.971,A -85,B 0,C 180,E1 -20791.097,E2 -20791.097} C_VEL
LIN {X 0,Y 366.677,Z 413.674,A -85,B 0,C 180,E1 -20792.197,E2 -20792.197} C_VEL
LIN {X 0,Y 365.979,Z 413.363,A -85,B 0,C 180,E1 -20793.303,E2 -20793.303} C_VEL
LIN {X 0,Y 364.911,Z 413.036,A -85,B 0,C 180,E1 -20794.418,E2 -20794.418} C_VEL
LIN {X 0,Y 363.542,Z 412.549,A -85,B 0,C 180,E1 -20795.547,E2 -20795.547} C_VEL
LIN {X 0,Y 361.233,Z 411.468,A -85,B 0,C 180,E1 -20797.151,E2 -20797.151} C_VEL
LIN {X 0,Y 357.743,Z 409.639,A -85,B 0,C 180,E1 -20799.042,E2 -20799.042} C_VEL
LIN {X 0,Y 353.989,Z 407.147,A -85,B 0,C 180,E1 -20800.813,E2 -20800.813} C_VEL
LIN {X 0,Y 349.069,Z 403.466,A -85,B 0,C 180,E1 -20802.795,E2 -20802.795} C_VEL
LIN {X 0,Y 344.795,Z 401.069,A -85,B 0,C 180,E1 -20804.158,E2 -20804.158} C_VEL
LIN {X 0,Y 339.951,Z 397.964,A -85,B 0,C 180,E1 -20805.59,E2 -20805.59} C_VEL
LIN {X 0,Y 334.336,Z 393.913,A -85,B 0,C 180,E1 -20807.115,E2 -20807.115} C_VEL
LIN {X 0,Y 328.782,Z 390.104,A -85,B 0,C 180,E1 -20808.45,E2 -20808.45} C_VEL
LIN {X 0,Y 321.606,Z 385.001,A -85,B 0,C 180,E1 -20810.006,E2 -20810.006} C_VEL
LIN {X 0,Y 316.305,Z 381.02,A -85,B 0,C 180,E1 -20811.063,E2 -20811.063} C_VEL
LIN {X 0,Y 308.345,Z 375.111,A -85,B 0,C 180,E1 -20812.472,E2 -20812.472} C_VEL
LIN {X 0,Y 299.992,Z 368.647,A -85,B 0,C 180,E1 -20813.757,E2 -20813.757} C_VEL
LIN {X 0,Y 288.176,Z 359.056,A -85,B 0,C 180,E1 -20815.33,E2 -20815.33} C_VEL
LIN {X 0,Y 274.288,Z 346.582,A -85,B 0,C 180,E1 -20817.151,E2 -20817.151} C_VEL
LIN {X 0,Y 260.388,Z 332.003,A -85,B 0,C 180,E1 -20819.195,E2 -20819.195} C_VEL
LIN {X 0,Y 251.199,Z 320.68,A -85,B 0,C 180,E1 -20820.751,E2 -20820.751} C_VEL
LIN {X 0,Y 241.961,Z 306.779,A -85,B 0,C 180,E1 -20822.551,E2 -20822.551} C_VEL
LIN {X 0,Y 234.655,Z 292.645,A -85,B 0,C 180,E1 -20824.218,E2 -20824.218} C_VEL
LIN {X 0,Y 228.476,Z 280.642,A -85,B 0,C 180,E1 -20825.741,E2 -20825.741} C_VEL
LIN {X 0,Y 220.909,Z 267.43,A -85,B 0,C 180,E1 -20827.708,E2 -20827.708} C_VEL
LIN {X 0,Y 216.379,Z 260.209,A -85,B 0,C 180,E1 -20828.95,E2 -20828.95} C_VEL
LIN {X 0,Y 214.256,Z 257.117,A -85,B 0,C 180,E1 -20829.555,E2 -20829.555} C_VEL
LIN {X 0,Y 213.822,Z 255.685,A -85,B 0,C 180,E1 -20829.912,E2 -20829.912} C_VEL
LIN {X 0,Y 213.721,Z 255.3,A -85,B 0,C 180,E1 -20830.86,E2 -20830.86} C_VEL
LIN {X 0,Y 213.727,Z 255.304,A -85,B 0,C 180,E1 -20833.673,E2 -20833.673} C_VEL
LIN {X 0,Y 213.809,Z 255.352,A -85,B 0,C 180,E1 -20836.349,E2 -20836.349} C_VEL
LIN {X 0,Y 213.792,Z 255.332,A -85,B 0,C 180,E1 -20839.12,E2 -20839.12} C_VEL
LIN {X 0,Y 213.753,Z 255.344,A -85,B 0,C 180,E1 -20843.715,E2 -20843.715} C_VEL
LIN {X 0,Y 213.768,Z 255.356,A -85,B 0,C 180,E1 -20848.264,E2 -20848.264} C_VEL
LIN {X 0,Y 213.824,Z 255.314,A -85,B 0,C 180,E1 -20852.604,E2 -20852.604} C_VEL
LIN {X 0,Y 213.818,Z 255.352,A -85,B 0,C 180,E1 -20856.975,E2 -20856.975} C_VEL
LIN {X 0,Y 213.942,Z 255.307,A -85,B 0,C 180,E1 -20862.805,E2 -20862.805} C_VEL
LIN {X 0,Y 213.953,Z 255.325,A -85,B 0,C 180,E1 -20866.708,E2 -20866.708} C_VEL
LIN {X 0,Y 214.141,Z 255.263,A -85,B 0,C 180,E1 -20870.556,E2 -20870.556} C_VEL
LIN {X 0,Y 214.208,Z 255.276,A -85,B 0,C 180,E1 -20872.46,E2 -20872.46} C_VEL
LIN {X 0,Y 214.445,Z 255.233,A -85,B 0,C 180,E1 -20878.123,E2 -20878.123} C_VEL
LIN {X 0,Y 214.546,Z 255.21,A -85,B 0,C 180,E1 -20880.001,E2 -20880.001} C_VEL
LIN {X 0,Y 214.444,Z 255.241,A -85,B 0,C 180,E1 -20881.879,E2 -20881.879} C_VEL
LIN {X 0,Y 214.184,Z 255.272,A -85,B 0,C 180,E1 -20887.543,E2 -20887.543} C_VEL
LIN {X 0,Y 213.997,Z 255.291,A -85,B 0,C 180,E1 -20891.365,E2 -20891.365} C_VEL
LIN {X 0,Y 213.91,Z 255.331,A -85,B 0,C 180,E1 -20895.24,E2 -20895.24} C_VEL
LIN {X 0,Y 213.826,Z 255.306,A -85,B 0,C 180,E1 -20899.19,E2 -20899.19} C_VEL
LIN {X 0,Y 213.849,Z 255.344,A -85,B 0,C 180,E1 -20903.228,E2 -20903.228} C_VEL
LIN {X 0,Y 213.831,Z 255.314,A -85,B 0,C 180,E1 -20907.451,E2 -20907.451} C_VEL
LIN {X 0,Y 213.769,Z 255.349,A -85,B 0,C 180,E1 -20911.738,E2 -20911.738} C_VEL
LIN {X 0,Y 213.746,Z 255.35,A -85,B 0,C 180,E1 -20916.289,E2 -20916.289} C_VEL
LIN {X 0,Y 213.713,Z 255.35,A -85,B 0,C 180,E1 -20921.126,E2 -20921.126} C_VEL
LIN {X 0,Y 213.765,Z 255.552,A -85,B 0,C 180,E1 -20925.651,E2 -20925.651} C_VEL
LIN {X 0,Y 215.26,Z 261.969,A -85,B 0,C 180,E1 -20930.112,E2 -20930.112} C_VEL
LIN {X 0,Y 215.561,Z 263.013,A -85,B 0,C 180,E1 -20930.563,E2 -20930.563} C_VEL
LIN {X 0,Y 217.785,Z 267.103,A -85,B 0,C 180,E1 -20931.254,E2 -20931.254} C_VEL
LIN {X 0,Y 224.661,Z 280.863,A -85,B 0,C 180,E1 -20933.177,E2 -20933.177} C_VEL
LIN {X 0,Y 231.106,Z 295.44,A -85,B 0,C 180,E1 -20934.899,E2 -20934.899} C_VEL
LIN {X 0,Y 232.579,Z 299.617,A -85,B 0,C 180,E1 -20935.305,E2 -20935.305} C_VEL
LIN {X 0,Y 236.044,Z 320.594,A -85,B 0,C 180,E1 -20936.632,E2 -20936.632} C_VEL
LIN {X 0,Y 234.085,Z 368.717,A -85,B 0,C 180,E1 -20938.088,E2 -20938.088} C_VEL
LIN {X 0,Y 233.13,Z 379.248,A -85,B 0,C 180,E1 -20938.585,E2 -20938.585} C_VEL
LIN {X 0,Y 232.653,Z 383.395,A -85,B 0,C 180,E1 -20938.816,E2 -20938.816} C_VEL
LIN {X 0,Y 231.287,Z 389.015,A -85,B 0,C 180,E1 -20939.114,E2 -20939.114} C_VEL
LIN {X 0,Y 227.334,Z 397.919,A -85,B 0,C 180,E1 -20939.566,E2 -20939.566} C_VEL
LIN {X 0,Y 223.163,Z 406.666,A -85,B 0,C 180,E1 -20940.195,E2 -20940.195} C_VEL
LIN {X 0,Y 221.453,Z 411.748,A -85,B 0,C 180,E1 -20940.771,E2 -20940.771} C_VEL
LIN {X 0,Y 218.819,Z 422.472,A -85,B 0,C 180,E1 -20942.504,E2 -20942.504} C_VEL
LIN {X 0,Y 216.655,Z 430.212,A -85,B 0,C 180,E1 -20944.029,E2 -20944.029} C_VEL
LIN {X 0,Y 213.92,Z 439.346,A -85,B 0,C 180,E1 -20946.268,E2 -20946.268} C_VEL
LIN {X 0,Y 212.16,Z 445.375,A -85,B 0,C 180,E1 -20948.055,E2 -20948.055} C_VEL
LIN {X 0,Y 210.023,Z 452.086,A -85,B 0,C 180,E1 -20950.45,E2 -20950.45} C_VEL
LIN {X 0,Y 208.632,Z 456.589,A -85,B 0,C 180,E1 -20952.352,E2 -20952.352} C_VEL
LIN {X 0,Y 206.804,Z 462.08,A -85,B 0,C 180,E1 -20955.234,E2 -20955.234} C_VEL
LIN {X 0,Y 205.578,Z 466.408,A -85,B 0,C 180,E1 -20958.164,E2 -20958.164} C_VEL
LIN {X 0,Y 205.023,Z 468.779,A -85,B 0,C 180,E1 -20960.131,E2 -20960.131} C_VEL
LIN {X 0,Y 204.627,Z 470.582,A -85,B 0,C 180,E1 -20962.104,E2 -20962.104} C_VEL
LIN {X 0,Y 204.319,Z 473.037,A -85,B 0,C 180,E1 -20966.055,E2 -20966.055} C_VEL
LIN {X 0,Y 204.331,Z 473.631,A -85,B 0,C 180,E1 -20968.029,E2 -20968.029} C_VEL
LIN {X 0,Y 204.438,Z 473.789,A -85,B 0,C 180,E1 -20970,E2 -20970} C_VEL
LIN {X 0,Y 204.331,Z 473.63,A -85,B 0,C 180,E1 -20971.971,E2 -20971.971} C_VEL
LIN {X 0,Y 204.299,Z 473.037,A -85,B 0,C 180,E1 -20973.945,E2 -20973.945} C_VEL
LIN {X 0,Y 204.608,Z 470.581,A -85,B 0,C 180,E1 -20977.897,E2 -20977.897} C_VEL
LIN {X 0,Y 205.28,Z 467.627,A -85,B 0,C 180,E1 -20980.853,E2 -20980.853} C_VEL
LIN {X 0,Y 206.311,Z 463.634,A -85,B 0,C 180,E1 -20983.795,E2 -20983.795} C_VEL
LIN {X 0,Y 207.941,Z 458.504,A -85,B 0,C 180,E1 -20986.695,E2 -20986.695} C_VEL
LIN {X 0,Y 209.605,Z 453.241,A -85,B 0,C 180,E1 -20989.082,E2 -20989.082} C_VEL
LIN {X 0,Y 211.722,Z 446.927,A -85,B 0,C 180,E1 -20991.416,E2 -20991.416} C_VEL
LIN {X 0,Y 213.442,Z 440.974,A -85,B 0,C 180,E1 -20993.274,E2 -20993.274} C_VEL
LIN {X 0,Y 215.511,Z 434.048,A -85,B 0,C 180,E1 -20995.084,E2 -20995.084} C_VEL
LIN {X 0,Y 217.889,Z 425.874,A -85,B 0,C 180,E1 -20996.844,E2 -20996.844} C_VEL
LIN {X 0,Y 220.103,Z 417.366,A -85,B 0,C 180,E1 -20998.357,E2 -20998.357} C_VEL
LIN {X 0,Y 222.093,Z 408.653,A -85,B 0,C 180,E1 -20999.633,E2 -20999.633} C_VEL
LIN {X 0,Y 223.932,Z 399.906,A -85,B 0,C 180,E1 -21000.664,E2 -21000.664} C_VEL
LIN {X 0,Y 225.595,Z 390.108,A -85,B 0,C 180,E1 -21001.585,E2 -21001.585} C_VEL
LIN {X 0,Y 226.995,Z 380.001,A -85,B 0,C 180,E1 -21002.295,E2 -21002.295} C_VEL
LIN {X 0,Y 228.03,Z 369.16,A -85,B 0,C 180,E1 -21002.829,E2 -21002.829} C_VEL
LIN {X 0,Y 229.606,Z 334.06,A -85,B 0,C 180,E1 -21003.927,E2 -21003.927} C_VEL
LIN {X 0,Y 230.054,Z 321.364,A -85,B 0,C 180,E1 -21004.321,E2 -21004.321} C_VEL
LIN {X 0,Y 226.819,Z 301.566,A -85,B 0,C 180,E1 -21005.627,E2 -21005.627} C_VEL
LIN {X 0,Y 221.014,Z 287.669,A -85,B 0,C 180,E1 -21007.257,E2 -21007.257} C_VEL
LIN {X 0,Y 214.43,Z 274.236,A -85,B 0,C 180,E1 -21009.163,E2 -21009.163} C_VEL
LIN {X 0,Y 210.052,Z 266.282,A -85,B 0,C 180,E1 -21010.484,E2 -21010.484} C_VEL
LIN {X 0,Y 208.176,Z 262.509,A -85,B 0,C 180,E1 -21011.181,E2 -21011.181} C_VEL
LIN {X 0,Y 207.297,Z 258.951,A -85,B 0,C 180,E1 -21013.579,E2 -21013.579} C_VEL
LIN {X 0,Y 206.665,Z 256.245,A -85,B 0,C 180,E1 -21015.728,E2 -21015.728} C_VEL
LIN {X 0,Y 206.662,Z 256.223,A -85,B 0,C 180,E1 -21019.748,E2 -21019.748} C_VEL
LIN {X 0,Y 206.701,Z 256.214,A -85,B 0,C 180,E1 -21024.688,E2 -21024.688} C_VEL
LIN {X 0,Y 206.709,Z 256.238,A -85,B 0,C 180,E1 -21029.336,E2 -21029.336} C_VEL
LIN {X 0,Y 206.733,Z 256.197,A -85,B 0,C 180,E1 -21033.771,E2 -21033.771} C_VEL
LIN {X 0,Y 206.758,Z 256.222,A -85,B 0,C 180,E1 -21038.042,E2 -21038.042} C_VEL
LIN {X 0,Y 206.869,Z 256.173,A -85,B 0,C 180,E1 -21042.195,E2 -21042.195} C_VEL
LIN {X 0,Y 206.883,Z 256.211,A -85,B 0,C 180,E1 -21046.242,E2 -21046.242} C_VEL
LIN {X 0,Y 207.079,Z 256.139,A -85,B 0,C 180,E1 -21050.229,E2 -21050.229} C_VEL
LIN {X 0,Y 207.052,Z 256.188,A -85,B 0,C 180,E1 -21054.154,E2 -21054.154} C_VEL
LIN {X 0,Y 207.38,Z 256.12,A -85,B 0,C 180,E1 -21058.057,E2 -21058.057} C_VEL
LIN {X 0,Y 207.512,Z 256.085,A -85,B 0,C 180,E1 -21059.999,E2 -21059.999} C_VEL
LIN {X 0,Y 207.382,Z 256.113,A -85,B 0,C 180,E1 -21061.941,E2 -21061.941} C_VEL
LIN {X 0,Y 207.148,Z 256.15,A -85,B 0,C 180,E1 -21067.799,E2 -21067.799} C_VEL
LIN {X 0,Y 206.924,Z 256.173,A -85,B 0,C 180,E1 -21071.757,E2 -21071.757} C_VEL
LIN {X 0,Y 206.867,Z 256.21,A -85,B 0,C 180,E1 -21075.77,E2 -21075.77} C_VEL
LIN {X 0,Y 206.761,Z 256.188,A -85,B 0,C 180,E1 -21079.87,E2 -21079.87} C_VEL
LIN {X 0,Y 206.745,Z 256.229,A -85,B 0,C 180,E1 -21084.073,E2 -21084.073} C_VEL
LIN {X 0,Y 206.735,Z 256.201,A -85,B 0,C 180,E1 -21088.419,E2 -21088.419} C_VEL
LIN {X 0,Y 206.703,Z 256.219,A -85,B 0,C 180,E1 -21092.955,E2 -21092.955} C_VEL
LIN {X 0,Y 206.723,Z 256.238,A -85,B 0,C 180,E1 -21097.729,E2 -21097.729} C_VEL
LIN {X 0,Y 206.721,Z 256.216,A -85,B 0,C 180,E1 -21101.588,E2 -21101.588} C_VEL
LIN {X 0,Y 206.659,Z 256.195,A -85,B 0,C 180,E1 -21105.573,E2 -21105.573} C_VEL
LIN {X 0,Y 206.693,Z 256.416,A -85,B 0,C 180,E1 -21108.333,E2 -21108.333} C_VEL
LIN {X 0,Y 206.924,Z 257.316,A -85,B 0,C 180,E1 -21108.717,E2 -21108.717} C_VEL
LIN {X 0,Y 208.491,Z 260.105,A -85,B 0,C 180,E1 -21109.258,E2 -21109.258} C_VEL
LIN {X 0,Y 209.698,Z 261.647,A -85,B 0,C 180,E1 -21109.612,E2 -21109.612} C_VEL
LIN {X 0,Y 218.537,Z 275.692,A -85,B 0,C 180,E1 -21112.145,E2 -21112.145} C_VEL
LIN {X 0,Y 227.137,Z 291.639,A -85,B 0,C 180,E1 -21114.435,E2 -21114.435} C_VEL
LIN {X 0,Y 236.106,Z 309.535,A -85,B 0,C 180,E1 -21116.629,E2 -21116.629} C_VEL
LIN {X 0,Y 244.228,Z 322.288,A -85,B 0,C 180,E1 -21118.318,E2 -21118.318} C_VEL
LIN {X 0,Y 252.153,Z 332.756,A -85,B 0,C 180,E1 -21119.77,E2 -21119.77} C_VEL
LIN {X 0,Y 264.707,Z 346.761,A -85,B 0,C 180,E1 -21121.777,E2 -21121.777} C_VEL
LIN {X 0,Y 276.81,Z 358.356,A -85,B 0,C 180,E1 -21123.503,E2 -21123.503} C_VEL
LIN {X 0,Y 287.005,Z 367.196,A -85,B 0,C 180,E1 -21124.961,E2 -21124.961} C_VEL
LIN {X 0,Y 298.597,Z 376.551,A -85,B 0,C 180,E1 -21126.623,E2 -21126.623} C_VEL
LIN {X 0,Y 307.017,Z 383.031,A -85,B 0,C 180,E1 -21127.984,E2 -21127.984} C_VEL
LIN {X 0,Y 315.179,Z 388.91,A -85,B 0,C 180,E1 -21129.475,E2 -21129.475} C_VEL
LIN {X 0,Y 321.83,Z 393.944,A -85,B 0,C 180,E1 -21130.879,E2 -21130.879} C_VEL
LIN {X 0,Y 329.427,Z 399.073,A -85,B 0,C 180,E1 -21132.622,E2 -21132.622} C_VEL
LIN {X 0,Y 335.758,Z 403.686,A -85,B 0,C 180,E1 -21134.332,E2 -21134.332} C_VEL
LIN {X 0,Y 340.744,Z 406.865,A -85,B 0,C 180,E1 -21135.785,E2 -21135.785} C_VEL
LIN {X 0,Y 345.686,Z 409.778,A -85,B 0,C 180,E1 -21137.383,E2 -21137.383} C_VEL
LIN {X 0,Y 350.428,Z 413.299,A -85,B 0,C 180,E1 -21139.328,E2 -21139.328} C_VEL
LIN {X 0,Y 355.181,Z 416.286,A -85,B 0,C 180,E1 -21141.627,E2 -21141.627} C_VEL
LIN {X 0,Y 357.989,Z 417.696,A -85,B 0,C 180,E1 -21143.235,E2 -21143.235} C_VEL
LIN {X 0,Y 359.991,Z 418.617,A -85,B 0,C 180,E1 -21144.651,E2 -21144.651} C_VEL
LIN {X 0,Y 362.148,Z 419.308,A -85,B 0,C 180,E1 -21146.662,E2 -21146.662} C_VEL
LIN {X 0,Y 362.821,Z 419.692,A -85,B 0,C 180,E1 -21147.78,E2 -21147.78} C_VEL
LIN {X 0,Y 363.188,Z 419.964,A -85,B 0,C 180,E1 -21148.891,E2 -21148.891} C_VEL
LIN {X 0,Y 363.419,Z 419.893,A -85,B 0,C 180,E1 -21150,E2 -21150} C_VEL
LIN {X 0,Y 363.198,Z 419.934,A -85,B 0,C 180,E1 -21151.109,E2 -21151.109} C_VEL
LIN {X 0,Y 362.833,Z 419.648,A -85,B 0,C 180,E1 -21152.22,E2 -21152.22} C_VEL
LIN {X 0,Y 362.118,Z 419.313,A -85,B 0,C 180,E1 -21153.338,E2 -21153.338} C_VEL
LIN {X 0,Y 359.983,Z 418.627,A -85,B 0,C 180,E1 -21155.336,E2 -21155.336} C_VEL
LIN {X 0,Y 357.957,Z 417.708,A -85,B 0,C 180,E1 -21156.765,E2 -21156.765} C_VEL
LIN {X 0,Y 355.188,Z 416.294,A -85,B 0,C 180,E1 -21158.381,E2 -21158.381} C_VEL
LIN {X 0,Y 350.42,Z 413.306,A -85,B 0,C 180,E1 -21160.664,E2 -21160.664} C_VEL
LIN {X 0,Y 345.675,Z 409.769,A -85,B 0,C 180,E1 -21162.609,E2 -21162.609} C_VEL
LIN {X 0,Y 340.27,Z 406.604,A -85,B 0,C 180,E1 -21164.35,E2 -21164.35} C_VEL
LIN {X 0,Y 333.094,Z 401.779,A -85,B 0,C 180,E1 -21166.407,E2 -21166.407} C_VEL
LIN {X 0,Y 327.613,Z 397.754,A -85,B 0,C 180,E1 -21167.828,E2 -21167.828} C_VEL
LIN {X 0,Y 320.441,Z 392.922,A -85,B 0,C 180,E1 -21169.426,E2 -21169.426} C_VEL
LIN {X 0,Y 311.989,Z 386.651,A -85,B 0,C 180,E1 -21171.126,E2 -21171.126} C_VEL
LIN {X 0,Y 304.251,Z 380.887,A -85,B 0,C 180,E1 -21172.488,E2 -21172.488} C_VEL
LIN {X 0,Y 295.132,Z 373.903,A -85,B 0,C 180,E1 -21173.88,E2 -21173.88} C_VEL
LIN {X 0,Y 279.902,Z 361.171,A -85,B 0,C 180,E1 -21176.051,E2 -21176.051} C_VEL
LIN {X 0,Y 269.107,Z 351.119,A -85,B 0,C 180,E1 -21177.589,E2 -21177.589} C_VEL
LIN {X 0,Y 255.786,Z 337.063,A -85,B 0,C 180,E1 -21179.617,E2 -21179.617} C_VEL
LIN {X 0,Y 246.396,Z 325.385,A -85,B 0,C 180,E1 -21181.266,E2 -21181.266} C_VEL
LIN {X 0,Y 236.995,Z 311.141,A -85,B 0,C 180,E1 -21183.171,E2 -21183.171} C_VEL
LIN {X 0,Y 229.121,Z 295.694,A -85,B 0,C 180,E1 -21185.056,E2 -21185.056} C_VEL
LIN {X 0,Y 222.395,Z 282.659,A -85,B 0,C 180,E1 -21186.805,E2 -21186.805} C_VEL
LIN {X 0,Y 215.648,Z 271.021,A -85,B 0,C 180,E1 -21188.654,E2 -21188.654} C_VEL
LIN {X 0,Y 211.094,Z 263.959,A -85,B 0,C 180,E1 -21189.963,E2 -21189.963} C_VEL
LIN {X 0,Y 209.034,Z 260.657,A -85,B 0,C 180,E1 -21190.588,E2 -21190.588} C_VEL
LIN {X 0,Y 207.199,Z 258.102,A -85,B 0,C 180,E1 -21191.15,E2 -21191.15} C_VEL
LIN {X 0,Y 206.719,Z 256.644,A -85,B 0,C 180,E1 -21191.515,E2 -21191.515} C_VEL
LIN {X 0,Y 206.631,Z 256.219,A -85,B 0,C 180,E1 -21192.133,E2 -21192.133} C_VEL
LIN {X 0,Y 206.713,Z 256.232,A -85,B 0,C 180,E1 -21197.16,E2 -21197.16} C_VEL
LIN {X 0,Y 206.758,Z 256.225,A -85,B 0,C 180,E1 -21201.426,E2 -21201.426} C_VEL
LIN {X 0,Y 206.729,Z 256.208,A -85,B 0,C 180,E1 -21204.696,E2 -21204.696} C_VEL
LIN {X 0,Y 206.706,Z 256.237,A -85,B 0,C 180,E1 -21209.337,E2 -21209.337} C_VEL
LIN {X 0,Y 206.728,Z 256.202,A -85,B 0,C 180,E1 -21213.773,E2 -21213.773} C_VEL
LIN {X 0,Y 206.737,Z 256.22,A -85,B 0,C 180,E1 -21218.042,E2 -21218.042} C_VEL
LIN {X 0,Y 206.871,Z 256.179,A -85,B 0,C 180,E1 -21222.198,E2 -21222.198} C_VEL
LIN {X 0,Y 206.895,Z 256.21,A -85,B 0,C 180,E1 -21226.245,E2 -21226.245} C_VEL
LIN {X 0,Y 207.099,Z 256.138,A -85,B 0,C 180,E1 -21230.232,E2 -21230.232} C_VEL
LIN {X 0,Y 207.066,Z 256.191,A -85,B 0,C 180,E1 -21234.157,E2 -21234.157} C_VEL
LIN {X 0,Y 207.382,Z 256.113,A -85,B 0,C 180,E1 -21238.059,E2 -21238.059} C_VEL
LIN {X 0,Y 207.512,Z 256.085,A -85,B 0,C 180,E1 -21240.001,E2 -21240.001} C_VEL
LIN {X 0,Y 207.38,Z 256.12,A -85,B 0,C 180,E1 -21241.943,E2 -21241.943} C_VEL
LIN {X 0,Y 207.128,Z 256.145,A -85,B 0,C 180,E1 -21247.801,E2 -21247.801} C_VEL
LIN {X 0,Y 206.921,Z 256.178,A -85,B 0,C 180,E1 -21251.76,E2 -21251.76} C_VEL
LIN {X 0,Y 206.843,Z 256.203,A -85,B 0,C 180,E1 -21255.774,E2 -21255.774} C_VEL
LIN {X 0,Y 206.858,Z 256.173,A -85,B 0,C 180,E1 -21257.955,E2 -21257.955} C_VEL
LIN {X 0,Y 206.787,Z 256.223,A -85,B 0,C 180,E1 -21263.417,E2 -21263.417} C_VEL
LIN {X 0,Y 206.739,Z 256.205,A -85,B 0,C 180,E1 -21268.421,E2 -21268.421} C_VEL
LIN {X 0,Y 206.701,Z 256.213,A -85,B 0,C 180,E1 -21272.958,E2 -21272.958} C_VEL
LIN {X 0,Y 206.684,Z 256.238,A -85,B 0,C 180,E1 -21277.74,E2 -21277.74} C_VEL
LIN {X 0,Y 206.643,Z 256.234,A -85,B 0,C 180,E1 -21281.563,E2 -21281.563} C_VEL
LIN {X 0,Y 206.686,Z 256.364,A -85,B 0,C 180,E1 -21284.433,E2 -21284.433} C_VEL
LIN {X 0,Y 208.085,Z 262.298,A -85,B 0,C 180,E1 -21288.721,E2 -21288.721} C_VEL
LIN {X 0,Y 208.956,Z 264.467,A -85,B 0,C 180,E1 -21289.181,E2 -21289.181} C_VEL
LIN {X 0,Y 213.551,Z 272.381,A -85,B 0,C 180,E1 -21290.568,E2 -21290.568} C_VEL
LIN {X 0,Y 221.156,Z 287.995,A -85,B 0,C 180,E1 -21292.784,E2 -21292.784} C_VEL
LIN {X 0,Y 226.905,Z 301.781,A -85,B 0,C 180,E1 -21294.397,E2 -21294.397} C_VEL
LIN {X 0,Y 230.14,Z 322.137,A -85,B 0,C 180,E1 -21295.722,E2 -21295.722} C_VEL
LIN {X 0,Y 228.044,Z 369.28,A -85,B 0,C 180,E1 -21297.177,E2 -21297.177} C_VEL
LIN {X 0,Y 226.921,Z 380.735,A -85,B 0,C 180,E1 -21297.748,E2 -21297.748} C_VEL
LIN {X 0,Y 225.038,Z 393.845,A -85,B 0,C 180,E1 -21298.721,E2 -21298.721} C_VEL
LIN {X 0,Y 222.758,Z 405.389,A -85,B 0,C 180,E1 -21299.944,E2 -21299.944} C_VEL
LIN {X 0,Y 221.453,Z 411.748,A -85,B 0,C 180,E1 -21300.771,E2 -21300.771} C_VEL
LIN {X 0,Y 219.668,Z 416.832,A -85,B 0,C 180,E1 -21301.41,E2 -21301.41} C_VEL
LIN {X 0,Y 215.026,Z 424.707,A -85,B 0,C 180,E1 -21302.437,E2 -21302.437} C_VEL
LIN {X 0,Y 210.275,Z 432.052,A -85,B 0,C 180,E1 -21303.697,E2 -21303.697} C_VEL
LIN {X 0,Y 208.352,Z 436.303,A -85,B 0,C 180,E1 -21304.689,E2 -21304.689} C_VEL
LIN {X 0,Y 205.95,Z 443.974,A -85,B 0,C 180,E1 -21306.895,E2 -21306.895} C_VEL
LIN {X 0,Y 203.797,Z 450.739,A -85,B 0,C 180,E1 -21309.3,E2 -21309.3} C_VEL
LIN {X 0,Y 201.84,Z 456.395,A -85,B 0,C 180,E1 -21311.737,E2 -21311.737} C_VEL
LIN {X 0,Y 199.905,Z 461.886,A -85,B 0,C 180,E1 -21314.712,E2 -21314.712} C_VEL
LIN {X 0,Y 198.603,Z 466.215,A -85,B 0,C 180,E1 -21317.742,E2 -21317.742} C_VEL
LIN {X 0,Y 198.001,Z 468.586,A -85,B 0,C 180,E1 -21319.777,E2 -21319.777} C_VEL
LIN {X 0,Y 197.578,Z 470.389,A -85,B 0,C 180,E1 -21321.82,E2 -21321.82} C_VEL
LIN {X 0,Y 197.242,Z 472.901,A -85,B 0,C 180,E1 -21326.107,E2 -21326.107} C_VEL
LIN {X 0,Y 197.239,Z 473.438,A -85,B 0,C 180,E1 -21327.958,E2 -21327.958} C_VEL
LIN {X 0,Y 197.34,Z 473.596,A -85,B 0,C 180,E1 -21330,E2 -21330} C_VEL
LIN {X 0,Y 197.237,Z 473.438,A -85,B 0,C 180,E1 -21332.042,E2 -21332.042} C_VEL
LIN {X 0,Y 197.21,Z 472.844,A -85,B 0,C 180,E1 -21334.087,E2 -21334.087} C_VEL
LIN {X 0,Y 197.544,Z 470.388,A -85,B 0,C 180,E1 -21338.181,E2 -21338.181} C_VEL
LIN {X 0,Y 198.27,Z 467.433,A -85,B 0,C 180,E1 -21341.242,E2 -21341.242} C_VEL
LIN {X 0,Y 199.384,Z 463.44,A -85,B 0,C 180,E1 -21344.285,E2 -21344.285} C_VEL
LIN {X 0,Y 201.127,Z 458.31,A -85,B 0,C 180,E1 -21347.278,E2 -21347.278} C_VEL
LIN {X 0,Y 202.892,Z 453.048,A -85,B 0,C 180,E1 -21349.739,E2 -21349.739} C_VEL
LIN {X 0,Y 205.067,Z 446.733,A -85,B 0,C 180,E1 -21352.147,E2 -21352.147} C_VEL
LIN {X 0,Y 207.413,Z 439.153,A -85,B 0,C 180,E1 -21354.524,E2 -21354.524} C_VEL
LIN {X 0,Y 210.303,Z 430.019,A -85,B 0,C 180,E1 -21356.817,E2 -21356.817} C_VEL
LIN {X 0,Y 213.525,Z 418.524,A -85,B 0,C 180,E1 -21359.044,E2 -21359.044} C_VEL
LIN {X 0,Y 215.938,Z 408.46,A -85,B 0,C 180,E1 -21360.566,E2 -21360.566} C_VEL
LIN {X 0,Y 217.86,Z 399.714,A -85,B 0,C 180,E1 -21361.615,E2 -21361.615} C_VEL
LIN {X 0,Y 219.589,Z 389.915,A -85,B 0,C 180,E1 -21362.553,E2 -21362.553} C_VEL
LIN {X 0,Y 221.079,Z 379.32,A -85,B 0,C 180,E1 -21363.307,E2 -21363.307} C_VEL
LIN {X 0,Y 222.06,Z 369.696,A -85,B 0,C 180,E1 -21363.791,E2 -21363.791} C_VEL
LIN {X 0,Y 223.448,Z 341.518,A -85,B 0,C 180,E1 -21364.703,E2 -21364.703} C_VEL
LIN {X 0,Y 224.195,Z 322.436,A -85,B 0,C 180,E1 -21365.301,E2 -21365.301} C_VEL
LIN {X 0,Y 221.223,Z 304.067,A -85,B 0,C 180,E1 -21366.566,E2 -21366.566} C_VEL
LIN {X 0,Y 215.872,Z 291.258,A -85,B 0,C 180,E1 -21368.147,E2 -21368.147} C_VEL
LIN {X 0,Y 208.497,Z 275.993,A -85,B 0,C 180,E1 -21370.416,E2 -21370.416} C_VEL
LIN {X 0,Y 202.967,Z 266.327,A -85,B 0,C 180,E1 -21372.199,E2 -21372.199} C_VEL
LIN {X 0,Y 200.861,Z 262.318,A -85,B 0,C 180,E1 -21373.019,E2 -21373.019} C_VEL
LIN {X 0,Y 200.347,Z 259.995,A -85,B 0,C 180,E1 -21374.554,E2 -21374.554} C_VEL
LIN {X 0,Y 199.605,Z 257.121,A -85,B 0,C 180,E1 -21377.052,E2 -21377.052} C_VEL
LIN {X 0,Y 199.613,Z 257.102,A -85,B 0,C 180,E1 -21380.767,E2 -21380.767} C_VEL
LIN {X 0,Y 199.613,Z 257.09,A -85,B 0,C 180,E1 -21385.712,E2 -21385.712} C_VEL
LIN {X 0,Y 199.695,Z 257.099,A -85,B 0,C 180,E1 -21388.135,E2 -21388.135} C_VEL
LIN {X 0,Y 199.687,Z 257.073,A -85,B 0,C 180,E1 -21392.771,E2 -21392.771} C_VEL
LIN {X 0,Y 199.739,Z 257.103,A -85,B 0,C 180,E1 -21397.228,E2 -21397.228} C_VEL
LIN {X 0,Y 199.796,Z 257.051,A -85,B 0,C 180,E1 -21401.758,E2 -21401.758} C_VEL
LIN {X 0,Y 199.822,Z 257.091,A -85,B 0,C 180,E1 -21405.746,E2 -21405.746} C_VEL
LIN {X 0,Y 200.023,Z 257.018,A -85,B 0,C 180,E1 -21409.881,E2 -21409.881} C_VEL
LIN {X 0,Y 200.013,Z 257.06,A -85,B 0,C 180,E1 -21413.948,E2 -21413.948} C_VEL
LIN {X 0,Y 200.319,Z 256.999,A -85,B 0,C 180,E1 -21417.988,E2 -21417.988} C_VEL
LIN {X 0,Y 200.476,Z 256.961,A -85,B 0,C 180,E1 -21419.999,E2 -21419.999} C_VEL
LIN {X 0,Y 200.029,Z 257.063,A -85,B 0,C 180,E1 -21424.028,E2 -21424.028} C_VEL
LIN {X 0,Y 200.095,Z 257.023,A -85,B 0,C 180,E1 -21428.075,E2 -21428.075} C_VEL
LIN {X 0,Y 199.874,Z 257.056,A -85,B 0,C 180,E1 -21432.178,E2 -21432.178} C_VEL
LIN {X 0,Y 199.804,Z 257.081,A -85,B 0,C 180,E1 -21436.342,E2 -21436.342} C_VEL
LIN {X 0,Y 199.68,Z 257.076,A -85,B 0,C 180,E1 -21440.606,E2 -21440.606} C_VEL
LIN {X 0,Y 199.663,Z 257.097,A -85,B 0,C 180,E1 -21444.984,E2 -21444.984} C_VEL
LIN {X 0,Y 199.663,Z 257.095,A -85,B 0,C 180,E1 -21449.523,E2 -21449.523} C_VEL
LIN {X 0,Y 199.656,Z 257.104,A -85,B 0,C 180,E1 -21452.348,E2 -21452.348} C_VEL
LIN {X 0,Y 199.651,Z 257.106,A -85,B 0,C 180,E1 -21456.756,E2 -21456.756} C_VEL
LIN {X 0,Y 199.676,Z 257.097,A -85,B 0,C 180,E1 -21459.311,E2 -21459.311} C_VEL
LIN {X 0,Y 199.66,Z 257.102,A -85,B 0,C 180,E1 -21462.337,E2 -21462.337} C_VEL
LIN {X 0,Y 199.633,Z 257.305,A -85,B 0,C 180,E1 -21466.518,E2 -21466.518} C_VEL
LIN {X 0,Y 199.845,Z 258.24,A -85,B 0,C 180,E1 -21466.944,E2 -21466.944} C_VEL
LIN {X 0,Y 201.435,Z 261.04,A -85,B 0,C 180,E1 -21467.538,E2 -21467.538} C_VEL
LIN {X 0,Y 202.682,Z 262.498,A -85,B 0,C 180,E1 -21467.931,E2 -21467.931} C_VEL
LIN {X 0,Y 205.028,Z 265.954,A -85,B 0,C 180,E1 -21468.682,E2 -21468.682} C_VEL
LIN {X 0,Y 213.818,Z 280.013,A -85,B 0,C 180,E1 -21471.331,E2 -21471.331} C_VEL
LIN {X 0,Y 222.284,Z 295.944,A -85,B 0,C 180,E1 -21473.698,E2 -21473.698} C_VEL
LIN {X 0,Y 231.179,Z 313.896,A -85,B 0,C 180,E1 -21475.976,E2 -21475.976} C_VEL
LIN {X 0,Y 239.378,Z 326.909,A -85,B 0,C 180,E1 -21477.754,E2 -21477.754} C_VEL
LIN {X 0,Y 247.245,Z 337.391,A -85,B 0,C 180,E1 -21479.254,E2 -21479.254} C_VEL
LIN {X 0,Y 260.344,Z 352.122,A -85,B 0,C 180,E1 -21481.422,E2 -21481.422} C_VEL
LIN {X 0,Y 271.504,Z 363.009,A -85,B 0,C 180,E1 -21483.154,E2 -21483.154} C_VEL
LIN {X 0,Y 282.578,Z 372.747,A -85,B 0,C 180,E1 -21484.885,E2 -21484.885} C_VEL
LIN {X 0,Y 295.72,Z 383.191,A -85,B 0,C 180,E1 -21486.897,E2 -21486.897} C_VEL
LIN {X 0,Y 304.238,Z 389.779,A -85,B 0,C 180,E1 -21488.309,E2 -21488.309} C_VEL
LIN {X 0,Y 310.755,Z 394.447,A -85,B 0,C 180,E1 -21489.504,E2 -21489.504} C_VEL
LIN {X 0,Y 316.464,Z 398.818,A -85,B 0,C 180,E1 -21490.702,E2 -21490.702} C_VEL
LIN {X 0,Y 324.308,Z 404.11,A -85,B 0,C 180,E1 -21492.459,E2 -21492.459} C_VEL
LIN {X 0,Y 329.858,Z 408.183,A -85,B 0,C 180,E1 -21493.92,E2 -21493.92} C_VEL
LIN {X 0,Y 335.135,Z 411.694,A -85,B 0,C 180,E1 -21495.425,E2 -21495.425} C_VEL
LIN {X 0,Y 341.104,Z 415.226,A -85,B 0,C 180,E1 -21497.308,E2 -21497.308} C_VEL
LIN {X 0,Y 344.202,Z 417.533,A -85,B 0,C 180,E1 -21498.54,E2 -21498.54} C_VEL
LIN {X 0,Y 346.373,Z 419.116,A -85,B 0,C 180,E1 -21499.478,E2 -21499.478} C_VEL
LIN {X 0,Y 349.07,Z 420.86,A -85,B 0,C 180,E1 -21500.731,E2 -21500.731} C_VEL
LIN {X 0,Y 351.441,Z 422.214,A -85,B 0,C 180,E1 -21501.953,E2 -21501.953} C_VEL
LIN {X 0,Y 353.802,Z 423.38,A -85,B 0,C 180,E1 -21503.313,E2 -21503.313} C_VEL
LIN {X 0,Y 355.263,Z 424.081,A -85,B 0,C 180,E1 -21504.323,E2 -21504.323} C_VEL
LIN {X 0,Y 356.693,Z 424.671,A -85,B 0,C 180,E1 -21505.48,E2 -21505.48} C_VEL
LIN {X 0,Y 357.866,Z 424.982,A -85,B 0,C 180,E1 -21506.622,E2 -21506.622} C_VEL
LIN {X 0,Y 358.657,Z 425.432,A -85,B 0,C 180,E1 -21507.931,E2 -21507.931} C_VEL
LIN {X 0,Y 359.181,Z 425.56,A -85,B 0,C 180,E1 -21510,E2 -21510} C_VEL
LIN {X 0,Y 358.653,Z 425.395,A -85,B 0,C 180,E1 -21512.053,E2 -21512.053} C_VEL
LIN {X 0,Y 357.83,Z 424.988,A -85,B 0,C 180,E1 -21513.378,E2 -21513.378} C_VEL
LIN {X 0,Y 356.668,Z 424.655,A -85,B 0,C 180,E1 -21514.521,E2 -21514.521} C_VEL
LIN {X 0,Y 353.786,Z 423.415,A -85,B 0,C 180,E1 -21516.665,E2 -21516.665} C_VEL
LIN {X 0,Y 351.429,Z 422.2,A -85,B 0,C 180,E1 -21518.047,E2 -21518.047} C_VEL
LIN {X 0,Y 348.961,Z 420.82,A -85,B 0,C 180,E1 -21519.307,E2 -21519.307} C_VEL
LIN {X 0,Y 346.351,Z 419.109,A -85,B 0,C 180,E1 -21520.523,E2 -21520.523} C_VEL
LIN {X 0,Y 343.322,Z 416.899,A -85,B 0,C 180,E1 -21521.812,E2 -21521.812} C_VEL
LIN {X 0,Y 339.373,Z 414.225,A -85,B 0,C 180,E1 -21523.271,E2 -21523.271} C_VEL
LIN {X 0,Y 334.363,Z 411.226,A -85,B 0,C 180,E1 -21524.791,E2 -21524.791} C_VEL
LIN {X 0,Y 327.997,Z 406.822,A -85,B 0,C 180,E1 -21526.585,E2 -21526.585} C_VEL
LIN {X 0,Y 321.721,Z 402.39,A -85,B 0,C 180,E1 -21528.148,E2 -21528.148} C_VEL
LIN {X 0,Y 313.834,Z 396.867,A -85,B 0,C 180,E1 -21529.859,E2 -21529.859} C_VEL
LIN {X 0,Y 308.489,Z 392.825,A -85,B 0,C 180,E1 -21530.925,E2 -21530.925} C_VEL
LIN {X 0,Y 301.607,Z 387.8,A -85,B 0,C 180,E1 -21532.145,E2 -21532.145} C_VEL
LIN {X 0,Y 291.684,Z 380.188,A -85,B 0,C 180,E1 -21533.712,E2 -21533.712} C_VEL
LIN {X 0,Y 276.67,Z 367.768,A -85,B 0,C 180,E1 -21536.028,E2 -21536.028} C_VEL
LIN {X 0,Y 265.037,Z 356.836,A -85,B 0,C 180,E1 -21537.851,E2 -21537.851} C_VEL
LIN {X 0,Y 251.788,Z 342.834,A -85,B 0,C 180,E1 -21539.952,E2 -21539.952} C_VEL
LIN {X 0,Y 241.871,Z 330.481,A -85,B 0,C 180,E1 -21541.749,E2 -21541.749} C_VEL
LIN {X 0,Y 232.302,Z 315.914,A -85,B 0,C 180,E1 -21543.763,E2 -21543.763} C_VEL
LIN {X 0,Y 224.466,Z 300.534,A -85,B 0,C 180,E1 -21545.713,E2 -21545.713} C_VEL
LIN {X 0,Y 218.362,Z 288.317,A -85,B 0,C 180,E1 -21547.376,E2 -21547.376} C_VEL
LIN {X 0,Y 211.267,Z 275.87,A -85,B 0,C 180,E1 -21549.407,E2 -21549.407} C_VEL
LIN {X 0,Y 204.742,Z 265.649,A -85,B 0,C 180,E1 -21551.403,E2 -21551.403} C_VEL
LIN {X 0,Y 201.957,Z 261.555,A -85,B 0,C 180,E1 -21552.301,E2 -21552.301} C_VEL
LIN {X 0,Y 200.15,Z 259.039,A -85,B 0,C 180,E1 -21552.904,E2 -21552.904} C_VEL
LIN {X 0,Y 199.696,Z 257.62,A -85,B 0,C 180,E1 -21553.256,E2 -21553.256} C_VEL
LIN {X 0,Y 199.615,Z 257.194,A -85,B 0,C 180,E1 -21553.638,E2 -21553.638} C_VEL
LIN {X 0,Y 199.663,Z 257.097,A -85,B 0,C 180,E1 -21558.028,E2 -21558.028} C_VEL
LIN {X 0,Y 199.677,Z 257.097,A -85,B 0,C 180,E1 -21560.744,E2 -21560.744} C_VEL
LIN {X 0,Y 199.63,Z 257.09,A -85,B 0,C 180,E1 -21565.718,E2 -21565.718} C_VEL
LIN {X 0,Y 199.694,Z 257.107,A -85,B 0,C 180,E1 -21568.137,E2 -21568.137} C_VEL
LIN {X 0,Y 199.682,Z 257.074,A -85,B 0,C 180,E1 -21572.772,E2 -21572.772} C_VEL
LIN {X 0,Y 199.713,Z 257.106,A -85,B 0,C 180,E1 -21577.227,E2 -21577.227} C_VEL
LIN {X 0,Y 199.794,Z 257.056,A -85,B 0,C 180,E1 -21581.76,E2 -21581.76} C_VEL
LIN {X 0,Y 199.836,Z 257.092,A -85,B 0,C 180,E1 -21585.749,E2 -21585.749} C_VEL
LIN {X 0,Y 200.022,Z 257.019,A -85,B 0,C 180,E1 -21589.883,E2 -21589.883} C_VEL
LIN {X 0,Y 200.027,Z 257.064,A -85,B 0,C 180,E1 -21593.951,E2 -21593.951} C_VEL
LIN {X 0,Y 200.321,Z 256.992,A -85,B 0,C 180,E1 -21597.991,E2 -21597.991} C_VEL
LIN {X 0,Y 200.476,Z 256.961,A -85,B 0,C 180,E1 -21600.001,E2 -21600.001} C_VEL
LIN {X 0,Y 200.022,Z 257.069,A -85,B 0,C 180,E1 -21604.031,E2 -21604.031} C_VEL
LIN {X 0,Y 200.076,Z 257.019,A -85,B 0,C 180,E1 -21608.078,E2 -21608.078} C_VEL
LIN {X 0,Y 199.87,Z 257.062,A -85,B 0,C 180,E1 -21612.181,E2 -21612.181} C_VEL
LIN {X 0,Y 199.788,Z 257.071,A -85,B 0,C 180,E1 -21616.346,E2 -21616.346} C_VEL
LIN {X 0,Y 199.687,Z 257.078,A -85,B 0,C 180,E1 -21620.608,E2 -21620.608} C_VEL
LIN {X 0,Y 199.738,Z 257.097,A -85,B 0,C 180,E1 -21623.818,E2 -21623.818} C_VEL
LIN {X 0,Y 199.71,Z 257.079,A -85,B 0,C 180,E1 -21628.385,E2 -21628.385} C_VEL
LIN {X 0,Y 199.673,Z 257.094,A -85,B 0,C 180,E1 -21632.356,E2 -21632.356} C_VEL
LIN {X 0,Y 199.626,Z 257.116,A -85,B 0,C 180,E1 -21636.764,E2 -21636.764} C_VEL
LIN {X 0,Y 199.61,Z 257.102,A -85,B 0,C 180,E1 -21639.329,E2 -21639.329} C_VEL
LIN {X 0,Y 199.646,Z 257.299,A -85,B 0,C 180,E1 -21643.263,E2 -21643.263} C_VEL
LIN {X 0,Y 200.709,Z 261.762,A -85,B 0,C 180,E1 -21646.72,E2 -21646.72} C_VEL
LIN {X 0,Y 201.017,Z 262.774,A -85,B 0,C 180,E1 -21647.087,E2 -21647.087} C_VEL
LIN {X 0,Y 203.28,Z 266.775,A -85,B 0,C 180,E1 -21647.901,E2 -21647.901} C_VEL
LIN {X 0,Y 209.547,Z 278.099,A -85,B 0,C 180,E1 -21649.918,E2 -21649.918} C_VEL
LIN {X 0,Y 216.609,Z 292.865,A -85,B 0,C 180,E1 -21652.071,E2 -21652.071} C_VEL
LIN {X 0,Y 221.374,Z 304.42,A -85,B 0,C 180,E1 -21653.477,E2 -21653.477} C_VEL
LIN {X 0,Y 224.245,Z 323.371,A -85,B 0,C 180,E1 -21654.744,E2 -21654.744} C_VEL
LIN {X 0,Y 222.137,Z 368.825,A -85,B 0,C 180,E1 -21656.174,E2 -21656.174} C_VEL
LIN {X 0,Y 221.026,Z 380.048,A -85,B 0,C 180,E1 -21656.74,E2 -21656.74} C_VEL
LIN {X 0,Y 219.193,Z 392.488,A -85,B 0,C 180,E1 -21657.653,E2 -21657.653} C_VEL
LIN {X 0,Y 216.653,Z 405.197,A -85,B 0,C 180,E1 -21659.005,E2 -21659.005} C_VEL
LIN {X 0,Y 214.556,Z 414.471,A -85,B 0,C 180,E1 -21660.302,E2 -21660.302} C_VEL
LIN {X 0,Y 212.209,Z 423.413,A -85,B 0,C 180,E1 -21661.84,E2 -21661.84} C_VEL
LIN {X 0,Y 209.683,Z 431.937,A -85,B 0,C 180,E1 -21663.634,E2 -21663.634} C_VEL
LIN {X 0,Y 208.352,Z 436.303,A -85,B 0,C 180,E1 -21664.689,E2 -21664.689} C_VEL
LIN {X 0,Y 206.442,Z 440.392,A -85,B 0,C 180,E1 -21665.75,E2 -21665.75} C_VEL
LIN {X 0,Y 201.705,Z 446.69,A -85,B 0,C 180,E1 -21667.453,E2 -21667.453} C_VEL
LIN {X 0,Y 197.049,Z 452.38,A -85,B 0,C 180,E1 -21669.369,E2 -21669.369} C_VEL
LIN {X 0,Y 195.313,Z 455.514,A -85,B 0,C 180,E1 -21670.742,E2 -21670.742} C_VEL
LIN {X 0,Y 193.034,Z 461.692,A -85,B 0,C 180,E1 -21674.154,E2 -21674.154} C_VEL
LIN {X 0,Y 191.648,Z 466.021,A -85,B 0,C 180,E1 -21677.289,E2 -21677.289} C_VEL
LIN {X 0,Y 190.996,Z 468.392,A -85,B 0,C 180,E1 -21679.398,E2 -21679.398} C_VEL
LIN {X 0,Y 190.528,Z 470.195,A -85,B 0,C 180,E1 -21681.515,E2 -21681.515} C_VEL
LIN {X 0,Y 190.165,Z 472.652,A -85,B 0,C 180,E1 -21685.761,E2 -21685.761} C_VEL
LIN {X 0,Y 190.149,Z 473.245,A -85,B 0,C 180,E1 -21687.882,E2 -21687.882} C_VEL
LIN {X 0,Y 190.243,Z 473.404,A -85,B 0,C 180,E1 -21690,E2 -21690} C_VEL
LIN {X 0,Y 190.12,Z 472.85,A -85,B 0,C 180,E1 -21693.529,E2 -21693.529} C_VEL
LIN {X 0,Y 190.231,Z 471.587,A -85,B 0,C 180,E1 -21696.363,E2 -21696.363} C_VEL
LIN {X 0,Y 190.502,Z 470.195,A -85,B 0,C 180,E1 -21698.486,E2 -21698.486} C_VEL
LIN {X 0,Y 191.283,Z 467.24,A -85,B 0,C 180,E1 -21701.658,E2 -21701.658} C_VEL
LIN {X 0,Y 192.471,Z 463.246,A -85,B 0,C 180,E1 -21704.809,E2 -21704.809} C_VEL
LIN {X 0,Y 194.337,Z 458.117,A -85,B 0,C 180,E1 -21707.902,E2 -21707.902} C_VEL
LIN {X 0,Y 196.214,Z 452.855,A -85,B 0,C 180,E1 -21710.44,E2 -21710.44} C_VEL
LIN {X 0,Y 198.131,Z 447.599,A -85,B 0,C 180,E1 -21712.542,E2 -21712.542} C_VEL
LIN {X 0,Y 200.42,Z 440.586,A -85,B 0,C 180,E1 -21714.885,E2 -21714.885} C_VEL
LIN {X 0,Y 202.707,Z 433.662,A -85,B 0,C 180,E1 -21716.79,E2 -21716.79} C_VEL
LIN {X 0,Y 205.272,Z 425.487,A -85,B 0,C 180,E1 -21718.641,E2 -21718.641} C_VEL
LIN {X 0,Y 207.696,Z 416.98,A -85,B 0,C 180,E1 -21720.221,E2 -21720.221} C_VEL
LIN {X 0,Y 209.84,Z 408.267,A -85,B 0,C 180,E1 -21721.555,E2 -21721.555} C_VEL
LIN {X 0,Y 212.021,Z 398.514,A -85,B 0,C 180,E1 -21722.733,E2 -21722.733} C_VEL
LIN {X 0,Y 213.866,Z 388.436,A -85,B 0,C 180,E1 -21723.679,E2 -21723.679} C_VEL
LIN {X 0,Y 215.326,Z 378.018,A -85,B 0,C 180,E1 -21724.409,E2 -21724.409} C_VEL
LIN {X 0,Y 216.295,Z 368.211,A -85,B 0,C 180,E1 -21724.888,E2 -21724.888} C_VEL
LIN {X 0,Y 218.415,Z 323.371,A -85,B 0,C 180,E1 -21726.337,E2 -21726.337} C_VEL
LIN {X 0,Y 215.604,Z 306.376,A -85,B 0,C 180,E1 -21727.579,E2 -21727.579} C_VEL
LIN {X 0,Y 210.349,Z 293.836,A -85,B 0,C 180,E1 -21729.219,E2 -21729.219} C_VEL
LIN {X 0,Y 203.798,Z 280.178,A -85,B 0,C 180,E1 -21731.351,E2 -21731.351} C_VEL
LIN {X 0,Y 198.452,Z 270.746,A -85,B 0,C 180,E1 -21733.17,E2 -21733.17} C_VEL
LIN {X 0,Y 195.363,Z 265.55,A -85,B 0,C 180,E1 -21734.28,E2 -21734.28} C_VEL
LIN {X 0,Y 193.577,Z 261.919,A -85,B 0,C 180,E1 -21735.113,E2 -21735.113} C_VEL
LIN {X 0,Y 192.54,Z 258.041,A -85,B 0,C 180,E1 -21738.289,E2 -21738.289} C_VEL
LIN {X 0,Y 192.589,Z 257.987,A -85,B 0,C 180,E1 -21743.401,E2 -21743.401} C_VEL
LIN {X 0,Y 192.61,Z 257.967,A -85,B 0,C 180,E1 -21747.059,E2 -21747.059} C_VEL
LIN {X 0,Y 192.662,Z 257.955,A -85,B 0,C 180,E1 -21751.69,E2 -21751.69} C_VEL
LIN {X 0,Y 192.707,Z 257.975,A -85,B 0,C 180,E1 -21756.348,E2 -21756.348} C_VEL
LIN {X 0,Y 192.731,Z 257.929,A -85,B 0,C 180,E1 -21761.458,E2 -21761.458} C_VEL
LIN {X 0,Y 192.75,Z 257.97,A -85,B 0,C 180,E1 -21765.212,E2 -21765.212} C_VEL
LIN {X 0,Y 192.946,Z 257.901,A -85,B 0,C 180,E1 -21769.566,E2 -21769.566} C_VEL
LIN {X 0,Y 192.976,Z 257.933,A -85,B 0,C 180,E1 -21773.726,E2 -21773.726} C_VEL
LIN {X 0,Y 193.261,Z 257.878,A -85,B 0,C 180,E1 -21777.915,E2 -21777.915} C_VEL
LIN {X 0,Y 193.441,Z 257.836,A -85,B 0,C 180,E1 -21779.999,E2 -21779.999} C_VEL
LIN {X 0,Y 192.975,Z 257.943,A -85,B 0,C 180,E1 -21784.176,E2 -21784.176} C_VEL
LIN {X 0,Y 193.041,Z 257.897,A -85,B 0,C 180,E1 -21788.372,E2 -21788.372} C_VEL
LIN {X 0,Y 192.802,Z 257.944,A -85,B 0,C 180,E1 -21792.632,E2 -21792.632} C_VEL
LIN {X 0,Y 192.757,Z 257.946,A -85,B 0,C 180,E1 -21796.958,E2 -21796.958} C_VEL
LIN {X 0,Y 192.615,Z 257.966,A -85,B 0,C 180,E1 -21801.399,E2 -21801.399} C_VEL
LIN {X 0,Y 192.646,Z 257.984,A -85,B 0,C 180,E1 -21804.212,E2 -21804.212} C_VEL
LIN {X 0,Y 192.642,Z 257.96,A -85,B 0,C 180,E1 -21808.888,E2 -21808.888} C_VEL
LIN {X 0,Y 192.596,Z 257.972,A -85,B 0,C 180,E1 -21813.185,E2 -21813.185} C_VEL
LIN {X 0,Y 192.598,Z 257.991,A -85,B 0,C 180,E1 -21818.339,E2 -21818.339} C_VEL
LIN {X 0,Y 192.596,Z 257.993,A -85,B 0,C 180,E1 -21823.129,E2 -21823.129} C_VEL
LIN {X 0,Y 192.635,Z 258.233,A -85,B 0,C 180,E1 -21824.632,E2 -21824.632} C_VEL
LIN {X 0,Y 192.919,Z 259.362,A -85,B 0,C 180,E1 -21825.054,E2 -21825.054} C_VEL
LIN {X 0,Y 194.339,Z 261.869,A -85,B 0,C 180,E1 -21825.622,E2 -21825.622} C_VEL
LIN {X 0,Y 195.806,Z 263.509,A -85,B 0,C 180,E1 -21826.125,E2 -21826.125} C_VEL
LIN {X 0,Y 197.958,Z 266.797,A -85,B 0,C 180,E1 -21826.886,E2 -21826.886} C_VEL
LIN {X 0,Y 203.873,Z 275.785,A -85,B 0,C 180,E1 -21828.848,E2 -21828.848} C_VEL
LIN {X 0,Y 210.209,Z 286.264,A -85,B 0,C 180,E1 -21830.805,E2 -21830.805} C_VEL
LIN {X 0,Y 218.652,Z 302.669,A -85,B 0,C 180,E1 -21833.262,E2 -21833.262} C_VEL
LIN {X 0,Y 226.007,Z 317.754,A -85,B 0,C 180,E1 -21835.226,E2 -21835.226} C_VEL
LIN {X 0,Y 234.32,Z 331.179,A -85,B 0,C 180,E1 -21837.118,E2 -21837.118} C_VEL
LIN {X 0,Y 242.692,Z 342.451,A -85,B 0,C 180,E1 -21838.779,E2 -21838.779} C_VEL
LIN {X 0,Y 254.842,Z 356.313,A -85,B 0,C 180,E1 -21840.91,E2 -21840.91} C_VEL
LIN {X 0,Y 265.406,Z 367.014,A -85,B 0,C 180,E1 -21842.713,E2 -21842.713} C_VEL
LIN {X 0,Y 276.274,Z 376.776,A -85,B 0,C 180,E1 -21844.56,E2 -21844.56} C_VEL
LIN {X 0,Y 290.368,Z 388.024,A -85,B 0,C 180,E1 -21846.886,E2 -21846.886} C_VEL
LIN {X 0,Y 300.184,Z 395.522,A -85,B 0,C 180,E1 -21848.532,E2 -21848.532} C_VEL
LIN {X 0,Y 307.914,Z 401.216,A -85,B 0,C 180,E1 -21849.979,E2 -21849.979} C_VEL
LIN {X 0,Y 314.999,Z 406.33,A -85,B 0,C 180,E1 -21851.482,E2 -21851.482} C_VEL
LIN {X 0,Y 321.423,Z 410.74,A -85,B 0,C 180,E1 -21852.992,E2 -21852.992} C_VEL
LIN {X 0,Y 327.816,Z 415.313,A -85,B 0,C 180,E1 -21854.738,E2 -21854.738} C_VEL
LIN {X 0,Y 334.134,Z 419.204,A -85,B 0,C 180,E1 -21856.622,E2 -21856.622} C_VEL
LIN {X 0,Y 338.079,Z 421.789,A -85,B 0,C 180,E1 -21858.002,E2 -21858.002} C_VEL
LIN {X 0,Y 342.605,Z 425.04,A -85,B 0,C 180,E1 -21859.942,E2 -21859.942} C_VEL
LIN {X 0,Y 347.433,Z 427.911,A -85,B 0,C 180,E1 -21862.382,E2 -21862.382} C_VEL
LIN {X 0,Y 350.41,Z 429.32,A -85,B 0,C 180,E1 -21864.245,E2 -21864.245} C_VEL
LIN {X 0,Y 352.331,Z 430.111,A -85,B 0,C 180,E1 -21865.822,E2 -21865.822} C_VEL
LIN {X 0,Y 353.137,Z 430.321,A -85,B 0,C 180,E1 -21866.577,E2 -21866.577} C_VEL
LIN {X 0,Y 353.875,Z 430.716,A -85,B 0,C 180,E1 -21867.724,E2 -21867.724} C_VEL
LIN {X 0,Y 354.286,Z 430.97,A -85,B 0,C 180,E1 -21868.863,E2 -21868.863} C_VEL
LIN {X 0,Y 354.548,Z 430.914,A -85,B 0,C 180,E1 -21870,E2 -21870} C_VEL
LIN {X 0,Y 354.292,Z 430.948,A -85,B 0,C 180,E1 -21871.137,E2 -21871.137} C_VEL
LIN {X 0,Y 353.904,Z 430.659,A -85,B 0,C 180,E1 -21872.276,E2 -21872.276} C_VEL
LIN {X 0,Y 352.339,Z 430.114,A -85,B 0,C 180,E1 -21874.196,E2 -21874.196} C_VEL
LIN {X 0,Y 350.357,Z 429.328,A -85,B 0,C 180,E1 -21875.756,E2 -21875.756} C_VEL
LIN {X 0,Y 347.44,Z 427.926,A -85,B 0,C 180,E1 -21877.626,E2 -21877.626} C_VEL
LIN {X 0,Y 342.601,Z 425.057,A -85,B 0,C 180,E1 -21880.054,E2 -21880.054} C_VEL
LIN {X 0,Y 338.028,Z 421.771,A -85,B 0,C 180,E1 -21882,E2 -21882} C_VEL
LIN {X 0,Y 334.133,Z 419.23,A -85,B 0,C 180,E1 -21883.378,E2 -21883.378} C_VEL
LIN {X 0,Y 327.814,Z 415.313,A -85,B 0,C 180,E1 -21885.26,E2 -21885.26} C_VEL
LIN {X 0,Y 322.769,Z 411.727,A -85,B 0,C 180,E1 -21886.656,E2 -21886.656} C_VEL
LIN {X 0,Y 316.921,Z 407.619,A -85,B 0,C 180,E1 -21888.087,E2 -21888.087} C_VEL
LIN {X 0,Y 309.691,Z 402.553,A -85,B 0,C 180,E1 -21889.651,E2 -21889.651} C_VEL
LIN {X 0,Y 304.332,Z 398.512,A -85,B 0,C 180,E1 -21890.73,E2 -21890.73} C_VEL
LIN {X 0,Y 296.003,Z 392.383,A -85,B 0,C 180,E1 -21892.186,E2 -21892.186} C_VEL
LIN {X 0,Y 281.411,Z 381.025,A -85,B 0,C 180,E1 -21894.586,E2 -21894.586} C_VEL
LIN {X 0,Y 269.457,Z 370.695,A -85,B 0,C 180,E1 -21896.606,E2 -21896.606} C_VEL
LIN {X 0,Y 260.163,Z 361.722,A -85,B 0,C 180,E1 -21898.199,E2 -21898.199} C_VEL
LIN {X 0,Y 249.721,Z 350.7,A -85,B 0,C 180,E1 -21899.972,E2 -21899.972} C_VEL
LIN {X 0,Y 238.276,Z 336.839,A -85,B 0,C 180,E1 -21902.067,E2 -21902.067} C_VEL
LIN {X 0,Y 228.702,Z 322.401,A -85,B 0,C 180,E1 -21904.13,E2 -21904.13} C_VEL
LIN {X 0,Y 221.659,Z 309.254,A -85,B 0,C 180,E1 -21905.897,E2 -21905.897} C_VEL
LIN {X 0,Y 214.784,Z 294.946,A -85,B 0,C 180,E1 -21907.838,E2 -21907.838} C_VEL
LIN {X 0,Y 207.359,Z 281.353,A -85,B 0,C 180,E1 -21910.062,E2 -21910.062} C_VEL
LIN {X 0,Y 200.208,Z 270.168,A -85,B 0,C 180,E1 -21912.349,E2 -21912.349} C_VEL
LIN {X 0,Y 197.812,Z 266.637,A -85,B 0,C 180,E1 -21913.162,E2 -21913.162} C_VEL
LIN {X 0,Y 195.624,Z 263.151,A -85,B 0,C 180,E1 -21913.944,E2 -21913.944} C_VEL
LIN {X 0,Y 193.42,Z 260.551,A -85,B 0,C 180,E1 -21914.714,E2 -21914.714} C_VEL
LIN {X 0,Y 192.714,Z 258.655,A -85,B 0,C 180,E1 -21915.138,E2 -21915.138} C_VEL
LIN {X 0,Y 192.594,Z 258.046,A -85,B 0,C 180,E1 -21915.607,E2 -21915.607} C_VEL
LIN {X 0,Y 192.587,Z 257.974,A -85,B 0,C 180,E1 -21920.026,E2 -21920.026} C_VEL
LIN {X 0,Y 192.599,Z 257.97,A -85,B 0,C 180,E1 -21924.28,E2 -21924.28} C_VEL
LIN {X 0,Y 192.598,Z 257.994,A -85,B 0,C 180,E1 -21929.28,E2 -21929.28} C_VEL
LIN {X 0,Y 192.659,Z 257.952,A -85,B 0,C 180,E1 -21931.692,E2 -21931.692} C_VEL
LIN {X 0,Y 192.684,Z 257.984,A -85,B 0,C 180,E1 -21936.347,E2 -21936.347} C_VEL
LIN {X 0,Y 192.729,Z 257.933,A -85,B 0,C 180,E1 -21941.46,E2 -21941.46} C_VEL
LIN {X 0,Y 192.763,Z 257.974,A -85,B 0,C 180,E1 -21945.215,E2 -21945.215} C_VEL
LIN {X 0,Y 192.945,Z 257.901,A -85,B 0,C 180,E1 -21949.568,E2 -21949.568} C_VEL
LIN {X 0,Y 193.041,Z 257.897,A -85,B 0,C 180,E1 -21951.628,E2 -21951.628} C_VEL
LIN {X 0,Y 193.263,Z 257.87,A -85,B 0,C 180,E1 -21957.917,E2 -21957.917} C_VEL
LIN {X 0,Y 193.441,Z 257.836,A -85,B 0,C 180,E1 -21960.001,E2 -21960.001} C_VEL
LIN {X 0,Y 192.968,Z 257.948,A -85,B 0,C 180,E1 -21964.178,E2 -21964.178} C_VEL
LIN {X 0,Y 193.027,Z 257.893,A -85,B 0,C 180,E1 -21968.375,E2 -21968.375} C_VEL
LIN {X 0,Y 192.797,Z 257.95,A -85,B 0,C 180,E1 -21972.635,E2 -21972.635} C_VEL
LIN {X 0,Y 192.747,Z 257.937,A -85,B 0,C 180,E1 -21976.961,E2 -21976.961} C_VEL
LIN {X 0,Y 192.629,Z 257.97,A -85,B 0,C 180,E1 -21981.399,E2 -21981.399} C_VEL
LIN {X 0,Y 192.666,Z 257.972,A -85,B 0,C 180,E1 -21984.226,E2 -21984.226} C_VEL
LIN {X 0,Y 192.646,Z 257.964,A -85,B 0,C 180,E1 -21988.89,E2 -21988.89} C_VEL
LIN {X 0,Y 192.598,Z 257.966,A -85,B 0,C 180,E1 -21993.187,E2 -21993.187} C_VEL
LIN {X 0,Y 192.554,Z 257.989,A -85,B 0,C 180,E1 -21998.353,E2 -21998.353} C_VEL
LIN {X 0,Y 192.572,Z 258.202,A -85,B 0,C 180,E1 -22001.921,E2 -22001.921} C_VEL
LIN {X 0,Y 193.577,Z 261.918,A -85,B 0,C 180,E1 -22004.887,E2 -22004.887} C_VEL
LIN {X 0,Y 195.661,Z 265.966,A -85,B 0,C 180,E1 -22005.825,E2 -22005.825} C_VEL
LIN {X 0,Y 200.004,Z 273.413,A -85,B 0,C 180,E1 -22007.37,E2 -22007.37} C_VEL
LIN {X 0,Y 206.126,Z 284.693,A -85,B 0,C 180,E1 -22009.415,E2 -22009.415} C_VEL
LIN {X 0,Y 213.413,Z 300.903,A -85,B 0,C 180,E1 -22011.742,E2 -22011.742} C_VEL
LIN {X 0,Y 215.986,Z 307.722,A -85,B 0,C 180,E1 -22012.554,E2 -22012.554} C_VEL
LIN {X 0,Y 218.41,Z 323.435,A -85,B 0,C 180,E1 -22013.665,E2 -22013.665} C_VEL
LIN {X 0,Y 216.29,Z 368.356,A -85,B 0,C 180,E1 -22015.114,E2 -22015.114} C_VEL
LIN {X 0,Y 215.183,Z 379.38,A -85,B 0,C 180,E1 -22015.675,E2 -22015.675} C_VEL
LIN {X 0,Y 213.651,Z 389.723,A -85,B 0,C 180,E1 -22016.424,E2 -22016.424} C_VEL
LIN {X 0,Y 211.444,Z 401.534,A -85,B 0,C 180,E1 -22017.591,E2 -22017.591} C_VEL
LIN {X 0,Y 208.751,Z 412.927,A -85,B 0,C 180,E1 -22019.108,E2 -22019.108} C_VEL
LIN {X 0,Y 205.972,Z 423.22,A -85,B 0,C 180,E1 -22020.907,E2 -22020.907} C_VEL
LIN {X 0,Y 203.327,Z 431.744,A -85,B 0,C 180,E1 -22022.743,E2 -22022.743} C_VEL
LIN {X 0,Y 200.968,Z 438.96,A -85,B 0,C 180,E1 -22024.635,E2 -22024.635} C_VEL
LIN {X 0,Y 198.449,Z 446.538,A -85,B 0,C 180,E1 -22027.073,E2 -22027.073} C_VEL
LIN {X 0,Y 196.692,Z 451.701,A -85,B 0,C 180,E1 -22029.065,E2 -22029.065} C_VEL
LIN {X 0,Y 195.313,Z 455.514,A -85,B 0,C 180,E1 -22030.742,E2 -22030.742} C_VEL
LIN {X 0,Y 193.643,Z 458.4,A -85,B 0,C 180,E1 -22032.183,E2 -22032.183} C_VEL
LIN {X 0,Y 191.163,Z 461.066,A -85,B 0,C 180,E1 -22033.594,E2 -22033.594} C_VEL
LIN {X 0,Y 185.273,Z 466.145,A -85,B 0,C 180,E1 -22037.097,E2 -22037.097} C_VEL
LIN {X 0,Y 184.035,Z 467.989,A -85,B 0,C 180,E1 -22038.79,E2 -22038.79} C_VEL
LIN {X 0,Y 183.499,Z 470.002,A -85,B 0,C 180,E1 -22041.188,E2 -22041.188} C_VEL
LIN {X 0,Y 183.08,Z 472.459,A -85,B 0,C 180,E1 -22045.597,E2 -22045.597} C_VEL
LIN {X 0,Y 183.048,Z 473.052,A -85,B 0,C 180,E1 -22047.8,E2 -22047.8} C_VEL
LIN {X 0,Y 183.15,Z 473.211,A -85,B 0,C 180,E1 -22050,E2 -22050} C_VEL
LIN {X 0,Y 183.035,Z 472.756,A -85,B 0,C 180,E1 -22053.301,E2 -22053.301} C_VEL
LIN {X 0,Y 183.149,Z 471.394,A -85,B 0,C 180,E1 -22056.61,E2 -22056.61} C_VEL
LIN {X 0,Y 183.454,Z 470.001,A -85,B 0,C 180,E1 -22058.815,E2 -22058.815} C_VEL
LIN {X 0,Y 184.316,Z 467.046,A -85,B 0,C 180,E1 -22062.106,E2 -22062.106} C_VEL
LIN {X 0,Y 185.578,Z 463.052,A -85,B 0,C 180,E1 -22065.373,E2 -22065.373} C_VEL
LIN {X 0,Y 187.572,Z 457.924,A -85,B 0,C 180,E1 -22068.571,E2 -22068.571} C_VEL
LIN {X 0,Y 189.574,Z 452.662,A -85,B 0,C 180,E1 -22071.19,E2 -22071.19} C_VEL
LIN {X 0,Y 191.764,Z 446.723,A -85,B 0,C 180,E1 -22073.617,E2 -22073.617} C_VEL
LIN {X 0,Y 193.967,Z 440.393,A -85,B 0,C 180,E1 -22075.772,E2 -22075.772} C_VEL
LIN {X 0,Y 196.391,Z 433.469,A -85,B 0,C 180,E1 -22077.724,E2 -22077.724} C_VEL
LIN {X 0,Y 199.059,Z 425.294,A -85,B 0,C 180,E1 -22079.622,E2 -22079.622} C_VEL
LIN {X 0,Y 201.582,Z 416.787,A -85,B 0,C 180,E1 -22081.239,E2 -22081.239} C_VEL
LIN {X 0,Y 203.815,Z 408.074,A -85,B 0,C 180,E1 -22082.601,E2 -22082.601} C_VEL
LIN {X 0,Y 206.096,Z 398.321,A -85,B 0,C 180,E1 -22083.798,E2 -22083.798} C_VEL
LIN {X 0,Y 207.767,Z 389.53,A -85,B 0,C 180,E1 -22084.66,E2 -22084.66} C_VEL
LIN {X 0,Y 209.4,Z 378.769,A -85,B 0,C 180,E1 -22085.447,E2 -22085.447} C_VEL
LIN {X 0,Y 210.454,Z 368.871,A -85,B 0,C 180,E1 -22085.957,E2 -22085.957} C_VEL
LIN {X 0,Y 212.03,Z 339.13,A -85,B 0,C 180,E1 -22086.952,E2 -22086.952} C_VEL
LIN {X 0,Y 212.63,Z 324.097,A -85,B 0,C 180,E1 -22087.453,E2 -22087.453} C_VEL
LIN {X 0,Y 210.213,Z 309.161,A -85,B 0,C 180,E1 -22088.591,E2 -22088.591} C_VEL
LIN {X 0,Y 204.623,Z 295.729,A -85,B 0,C 180,E1 -22090.445,E2 -22090.445} C_VEL
LIN {X 0,Y 198.683,Z 283.461,A -85,B 0,C 180,E1 -22092.496,E2 -22092.496} C_VEL
LIN {X 0,Y 193.664,Z 274.535,A -85,B 0,C 180,E1 -22094.313,E2 -22094.313} C_VEL
LIN {X 0,Y 191.369,Z 270.545,A -85,B 0,C 180,E1 -22095.19,E2 -22095.19} C_VEL
LIN {X 0,Y 188.934,Z 266.392,A -85,B 0,C 180,E1 -22096.155,E2 -22096.155} C_VEL
LIN {X 0,Y 186.471,Z 262.406,A -85,B 0,C 180,E1 -22097.206,E2 -22097.206} C_VEL
LIN {X 0,Y 186.022,Z 261.12,A -85,B 0,C 180,E1 -22097.773,E2 -22097.773} C_VEL
LIN {X 0,Y 185.476,Z 258.888,A -85,B 0,C 180,E1 -22099.896,E2 -22099.896} C_VEL
LIN {X 0,Y 185.51,Z 258.878,A -85,B 0,C 180,E1 -22102.71,E2 -22102.71} C_VEL
LIN {X 0,Y 185.544,Z 258.857,A -85,B 0,C 180,E1 -22107.974,E2 -22107.974} C_VEL
LIN {X 0,Y 185.582,Z 258.851,A -85,B 0,C 180,E1 -22110.576,E2 -22110.576} C_VEL
LIN {X 0,Y 185.589,Z 258.845,A -85,B 0,C 180,E1 -22115.381,E2 -22115.381} C_VEL
LIN {X 0,Y 185.674,Z 258.808,A -85,B 0,C 180,E1 -22121.134,E2 -22121.134} C_VEL
LIN {X 0,Y 185.683,Z 258.842,A -85,B 0,C 180,E1 -22124.635,E2 -22124.635} C_VEL
LIN {X 0,Y 185.889,Z 258.78,A -85,B 0,C 180,E1 -22129.418,E2 -22129.418} C_VEL
LIN {X 0,Y 185.939,Z 258.803,A -85,B 0,C 180,E1 -22133.488,E2 -22133.488} C_VEL
LIN {X 0,Y 186.205,Z 258.757,A -85,B 0,C 180,E1 -22137.836,E2 -22137.836} C_VEL
LIN {X 0,Y 186.404,Z 258.712,A -85,B 0,C 180,E1 -22139.999,E2 -22139.999} C_VEL
LIN {X 0,Y 185.922,Z 258.823,A -85,B 0,C 180,E1 -22144.335,E2 -22144.335} C_VEL
LIN {X 0,Y 185.986,Z 258.771,A -85,B 0,C 180,E1 -22148.692,E2 -22148.692} C_VEL
LIN {X 0,Y 185.729,Z 258.833,A -85,B 0,C 180,E1 -22153.122,E2 -22153.122} C_VEL
LIN {X 0,Y 185.689,Z 258.816,A -85,B 0,C 180,E1 -22157.624,E2 -22157.624} C_VEL
LIN {X 0,Y 185.576,Z 258.857,A -85,B 0,C 180,E1 -22162.253,E2 -22162.253} C_VEL
LIN {X 0,Y 185.556,Z 258.833,A -85,B 0,C 180,E1 -22167.032,E2 -22167.032} C_VEL
LIN {X 0,Y 185.576,Z 258.847,A -85,B 0,C 180,E1 -22169.492,E2 -22169.492} C_VEL
LIN {X 0,Y 185.518,Z 258.846,A -85,B 0,C 180,E1 -22174.627,E2 -22174.627} C_VEL
LIN {X 0,Y 185.566,Z 258.868,A -85,B 0,C 180,E1 -22177.313,E2 -22177.313} C_VEL
LIN {X 0,Y 185.526,Z 258.943,A -85,B 0,C 180,E1 -22182.222,E2 -22182.222} C_VEL
LIN {X 0,Y 185.726,Z 259.842,A -85,B 0,C 180,E1 -22182.777,E2 -22182.777} C_VEL
LIN {X 0,Y 187.272,Z 262.667,A -85,B 0,C 180,E1 -22183.495,E2 -22183.495} C_VEL
LIN {X 0,Y 188.908,Z 264.416,A -85,B 0,C 180,E1 -22184.113,E2 -22184.113} C_VEL
LIN {X 0,Y 190.895,Z 267.575,A -85,B 0,C 180,E1 -22184.894,E2 -22184.894} C_VEL
LIN {X 0,Y 192.321,Z 269.552,A -85,B 0,C 180,E1 -22185.424,E2 -22185.424} C_VEL
LIN {X 0,Y 199.228,Z 279.915,A -85,B 0,C 180,E1 -22187.859,E2 -22187.859} C_VEL
LIN {X 0,Y 206.266,Z 291.871,A -85,B 0,C 180,E1 -22190.15,E2 -22190.15} C_VEL
LIN {X 0,Y 213.769,Z 306.833,A -85,B 0,C 180,E1 -22192.445,E2 -22192.445} C_VEL
LIN {X 0,Y 221.102,Z 322.035,A -85,B 0,C 180,E1 -22194.5,E2 -22194.5} C_VEL
LIN {X 0,Y 229.469,Z 335.71,A -85,B 0,C 180,E1 -22196.493,E2 -22196.493} C_VEL
LIN {X 0,Y 238.005,Z 347.344,A -85,B 0,C 180,E1 -22198.258,E2 -22198.258} C_VEL
LIN {X 0,Y 249.18,Z 360.335,A -85,B 0,C 180,E1 -22200.347,E2 -22200.347} C_VEL
LIN {X 0,Y 261.022,Z 372.547,A -85,B 0,C 180,E1 -22202.581,E2 -22202.581} C_VEL
LIN {X 0,Y 272.195,Z 382.604,A -85,B 0,C 180,E1 -22204.645,E2 -22204.645} C_VEL
LIN {X 0,Y 286.092,Z 393.576,A -85,B 0,C 180,E1 -22207.101,E2 -22207.101} C_VEL
LIN {X 0,Y 298.882,Z 403.16,A -85,B 0,C 180,E1 -22209.347,E2 -22209.347} C_VEL
LIN {X 0,Y 305.406,Z 408.062,A -85,B 0,C 180,E1 -22210.644,E2 -22210.644} C_VEL
LIN {X 0,Y 313.306,Z 413.536,A -85,B 0,C 180,E1 -22212.369,E2 -22212.369} C_VEL
LIN {X 0,Y 318.537,Z 417.291,A -85,B 0,C 180,E1 -22213.685,E2 -22213.685} C_VEL
LIN {X 0,Y 325.256,Z 421.856,A -85,B 0,C 180,E1 -22215.56,E2 -22215.56} C_VEL
LIN {X 0,Y 331.233,Z 425.475,A -85,B 0,C 180,E1 -22217.422,E2 -22217.422} C_VEL
LIN {X 0,Y 336.068,Z 428.991,A -85,B 0,C 180,E1 -22219.38,E2 -22219.38} C_VEL
LIN {X 0,Y 338.429,Z 430.546,A -85,B 0,C 180,E1 -22220.437,E2 -22220.437} C_VEL
LIN {X 0,Y 340.969,Z 432.092,A -85,B 0,C 180,E1 -22221.704,E2 -22221.704} C_VEL
LIN {X 0,Y 343.237,Z 433.284,A -85,B 0,C 180,E1 -22222.943,E2 -22222.943} C_VEL
LIN {X 0,Y 345.85,Z 434.526,A -85,B 0,C 180,E1 -22224.692,E2 -22224.692} C_VEL
LIN {X 0,Y 347.981,Z 435.278,A -85,B 0,C 180,E1 -22226.526,E2 -22226.526} C_VEL
LIN {X 0,Y 348.778,Z 435.656,A -85,B 0,C 180,E1 -22227.69,E2 -22227.69} C_VEL
LIN {X 0,Y 349.197,Z 435.926,A -85,B 0,C 180,E1 -22228.847,E2 -22228.847} C_VEL
LIN {X 0,Y 349.477,Z 435.882,A -85,B 0,C 180,E1 -22230,E2 -22230} C_VEL
LIN {X 0,Y 349.214,Z 435.895,A -85,B 0,C 180,E1 -22231.153,E2 -22231.153} C_VEL
LIN {X 0,Y 348.792,Z 435.617,A -85,B 0,C 180,E1 -22232.31,E2 -22232.31} C_VEL
LIN {X 0,Y 347.955,Z 435.266,A -85,B 0,C 180,E1 -22233.474,E2 -22233.474} C_VEL
LIN {X 0,Y 345.854,Z 434.555,A -85,B 0,C 180,E1 -22235.315,E2 -22235.315} C_VEL
LIN {X 0,Y 343.194,Z 433.284,A -85,B 0,C 180,E1 -22237.058,E2 -22237.058} C_VEL
LIN {X 0,Y 340.925,Z 432.05,A -85,B 0,C 180,E1 -22238.317,E2 -22238.317} C_VEL
LIN {X 0,Y 338.407,Z 430.536,A -85,B 0,C 180,E1 -22239.564,E2 -22239.564} C_VEL
LIN {X 0,Y 334.447,Z 427.811,A -85,B 0,C 180,E1 -22241.327,E2 -22241.327} C_VEL
LIN {X 0,Y 331.24,Z 425.486,A -85,B 0,C 180,E1 -22242.584,E2 -22242.584} C_VEL
LIN {X 0,Y 325.225,Z 421.87,A -85,B 0,C 180,E1 -22244.442,E2 -22244.442} C_VEL
LIN {X 0,Y 318.538,Z 417.276,A -85,B 0,C 180,E1 -22246.316,E2 -22246.316} C_VEL
LIN {X 0,Y 313.312,Z 413.538,A -85,B 0,C 180,E1 -22247.635,E2 -22247.635} C_VEL
LIN {X 0,Y 305.405,Z 408.064,A -85,B 0,C 180,E1 -22249.355,E2 -22249.355} C_VEL
LIN {X 0,Y 298.828,Z 403.134,A -85,B 0,C 180,E1 -22250.657,E2 -22250.657} C_VEL
LIN {X 0,Y 286.093,Z 393.57,A -85,B 0,C 180,E1 -22252.9,E2 -22252.9} C_VEL
LIN {X 0,Y 274.978,Z 384.835,A -85,B 0,C 180,E1 -22254.864,E2 -22254.864} C_VEL
LIN {X 0,Y 265.107,Z 376.316,A -85,B 0,C 180,E1 -22256.66,E2 -22256.66} C_VEL
LIN {X 0,Y 255.876,Z 367.402,A -85,B 0,C 180,E1 -22258.386,E2 -22258.386} C_VEL
LIN {X 0,Y 245.717,Z 356.446,A -85,B 0,C 180,E1 -22260.299,E2 -22260.299} C_VEL
LIN {X 0,Y 233.93,Z 342.101,A -85,B 0,C 180,E1 -22262.553,E2 -22262.553} C_VEL
LIN {X 0,Y 224.554,Z 327.98,A -85,B 0,C 180,E1 -22264.642,E2 -22264.642} C_VEL
LIN {X 0,Y 218.047,Z 316.135,A -85,B 0,C 180,E1 -22266.315,E2 -22266.315} C_VEL
LIN {X 0,Y 210.128,Z 299.344,A -85,B 0,C 180,E1 -22268.649,E2 -22268.649} C_VEL
LIN {X 0,Y 202.995,Z 286.065,A -85,B 0,C 180,E1 -22270.896,E2 -22270.896} C_VEL
LIN {X 0,Y 195.853,Z 274.763,A -85,B 0,C 180,E1 -22273.302,E2 -22273.302} C_VEL
LIN {X 0,Y 190.992,Z 267.679,A -85,B 0,C 180,E1 -22275.071,E2 -22275.071} C_VEL
LIN {X 0,Y 188.805,Z 264.217,A -85,B 0,C 180,E1 -22275.93,E2 -22275.93} C_VEL
LIN {X 0,Y 186.398,Z 261.445,A -85,B 0,C 180,E1 -22276.859,E2 -22276.859} C_VEL
LIN {X 0,Y 185.651,Z 259.475,A -85,B 0,C 180,E1 -22277.355,E2 -22277.355} C_VEL
LIN {X 0,Y 185.532,Z 258.906,A -85,B 0,C 180,E1 -22277.931,E2 -22277.931} C_VEL
LIN {X 0,Y 185.557,Z 258.869,A -85,B 0,C 180,E1 -22282.701,E2 -22282.701} C_VEL
LIN {X 0,Y 185.539,Z 258.866,A -85,B 0,C 180,E1 -22287.976,E2 -22287.976} C_VEL
LIN {X 0,Y 185.579,Z 258.845,A -85,B 0,C 180,E1 -22290.578,E2 -22290.578} C_VEL
LIN {X 0,Y 185.578,Z 258.856,A -85,B 0,C 180,E1 -22295.383,E2 -22295.383} C_VEL
LIN {X 0,Y 185.672,Z 258.811,A -85,B 0,C 180,E1 -22301.136,E2 -22301.136} C_VEL
LIN {X 0,Y 185.719,Z 258.848,A -85,B 0,C 180,E1 -22304.641,E2 -22304.641} C_VEL
LIN {X 0,Y 185.888,Z 258.779,A -85,B 0,C 180,E1 -22309.418,E2 -22309.418} C_VEL
LIN {X 0,Y 185.952,Z 258.81,A -85,B 0,C 180,E1 -22313.491,E2 -22313.491} C_VEL
LIN {X 0,Y 186.207,Z 258.749,A -85,B 0,C 180,E1 -22317.838,E2 -22317.838} C_VEL
LIN {X 0,Y 186.404,Z 258.712,A -85,B 0,C 180,E1 -22320.001,E2 -22320.001} C_VEL
LIN {X 0,Y 185.914,Z 258.826,A -85,B 0,C 180,E1 -22324.337,E2 -22324.337} C_VEL
LIN {X 0,Y 185.976,Z 258.768,A -85,B 0,C 180,E1 -22328.695,E2 -22328.695} C_VEL
LIN {X 0,Y 185.723,Z 258.839,A -85,B 0,C 180,E1 -22333.125,E2 -22333.125} C_VEL
LIN {X 0,Y 185.685,Z 258.81,A -85,B 0,C 180,E1 -22337.627,E2 -22337.627} C_VEL
LIN {X 0,Y 185.593,Z 258.86,A -85,B 0,C 180,E1 -22342.253,E2 -22342.253} C_VEL
LIN {X 0,Y 185.562,Z 258.831,A -85,B 0,C 180,E1 -22347.033,E2 -22347.033} C_VEL
LIN {X 0,Y 185.579,Z 258.853,A -85,B 0,C 180,E1 -22349.494,E2 -22349.494} C_VEL
LIN {X 0,Y 185.501,Z 258.848,A -85,B 0,C 180,E1 -22354.633,E2 -22354.633} C_VEL
LIN {X 0,Y 185.51,Z 258.878,A -85,B 0,C 180,E1 -22357.314,E2 -22357.314} C_VEL
LIN {X 0,Y 185.495,Z 259.085,A -85,B 0,C 180,E1 -22360.428,E2 -22360.428} C_VEL
LIN {X 0,Y 186.148,Z 261.538,A -85,B 0,C 180,E1 -22362.502,E2 -22362.502} C_VEL
LIN {X 0,Y 187.515,Z 264.44,A -85,B 0,C 180,E1 -22363.288,E2 -22363.288} C_VEL
LIN {X 0,Y 189.965,Z 268.057,A -85,B 0,C 180,E1 -22364.254,E2 -22364.254} C_VEL
LIN {X 0,Y 196.021,Z 278.67,A -85,B 0,C 180,E1 -22366.556,E2 -22366.556} C_VEL
LIN {X 0,Y 201.527,Z 289.05,A -85,B 0,C 180,E1 -22368.496,E2 -22368.496} C_VEL
LIN {X 0,Y 207.9,Z 303.368,A -85,B 0,C 180,E1 -22370.649,E2 -22370.649} C_VEL
LIN {X 0,Y 210.575,Z 310.56,A -85,B 0,C 180,E1 -22371.546,E2 -22371.546} C_VEL
LIN {X 0,Y 212.687,Z 324.619,A -85,B 0,C 180,E1 -22372.58,E2 -22372.58} C_VEL
LIN {X 0,Y 210.457,Z 368.938,A -85,B 0,C 180,E1 -22374.044,E2 -22374.044} C_VEL
LIN {X 0,Y 209.178,Z 380.727,A -85,B 0,C 180,E1 -22374.675,E2 -22374.675} C_VEL
LIN {X 0,Y 206.919,Z 394.295,A -85,B 0,C 180,E1 -22375.768,E2 -22375.768} C_VEL
LIN {X 0,Y 204.607,Z 404.811,A -85,B 0,C 180,E1 -22376.956,E2 -22376.956} C_VEL
LIN {X 0,Y 202.33,Z 414.085,A -85,B 0,C 180,E1 -22378.307,E2 -22378.307} C_VEL
LIN {X 0,Y 199.779,Z 423.027,A -85,B 0,C 180,E1 -22379.914,E2 -22379.914} C_VEL
LIN {X 0,Y 197.037,Z 431.551,A -85,B 0,C 180,E1 -22381.797,E2 -22381.797} C_VEL
LIN {X 0,Y 194.552,Z 438.766,A -85,B 0,C 180,E1 -22383.735,E2 -22383.735} C_VEL
LIN {X 0,Y 192.387,Z 444.968,A -85,B 0,C 180,E1 -22385.734,E2 -22385.734} C_VEL
LIN {X 0,Y 190.055,Z 451.507,A -85,B 0,C 180,E1 -22388.298,E2 -22388.298} C_VEL
LIN {X 0,Y 188.322,Z 456.008,A -85,B 0,C 180,E1 -22390.375,E2 -22390.375} C_VEL
LIN {X 0,Y 186.187,Z 461.499,A -85,B 0,C 180,E1 -22393.555,E2 -22393.555} C_VEL
LIN {X 0,Y 184.708,Z 465.828,A -85,B 0,C 180,E1 -22396.803,E2 -22396.803} C_VEL
LIN {X 0,Y 184.035,Z 467.989,A -85,B 0,C 180,E1 -22398.79,E2 -22398.79} C_VEL
LIN {X 0,Y 182.945,Z 469.639,A -85,B 0,C 180,E1 -22400.529,E2 -22400.529} C_VEL
LIN {X 0,Y 179.665,Z 471.582,A -85,B 0,C 180,E1 -22403.422,E2 -22403.422} C_VEL
LIN {X 0,Y 177.102,Z 472.492,A -85,B 0,C 180,E1 -22405.838,E2 -22405.838} C_VEL
LIN {X 0,Y 176.045,Z 472.869,A -85,B 0,C 180,E1 -22407.739,E2 -22407.739} C_VEL
LIN {X 0,Y 175.968,Z 472.907,A -85,B 0,C 180,E1 -22408.385,E2 -22408.385} C_VEL
LIN {X 0,Y 176.058,Z 473.018,A -85,B 0,C 180,E1 -22410,E2 -22410} C_VEL
LIN {X 0,Y 175.95,Z 472.666,A -85,B 0,C 180,E1 -22413.037,E2 -22413.037} C_VEL
LIN {X 0,Y 176.092,Z 471.201,A -85,B 0,C 180,E1 -22416.877,E2 -22416.877} C_VEL
LIN {X 0,Y 176.424,Z 469.808,A -85,B 0,C 180,E1 -22419.169,E2 -22419.169} C_VEL
LIN {X 0,Y 177.348,Z 466.853,A -85,B 0,C 180,E1 -22422.589,E2 -22422.589} C_VEL
LIN {X 0,Y 178.71,Z 462.858,A -85,B 0,C 180,E1 -22425.979,E2 -22425.979} C_VEL
LIN {X 0,Y 180.832,Z 457.73,A -85,B 0,C 180,E1 -22429.29,E2 -22429.29} C_VEL
LIN {X 0,Y 182.968,Z 452.469,A -85,B 0,C 180,E1 -22431.994,E2 -22431.994} C_VEL
LIN {X 0,Y 185.4,Z 446.151,A -85,B 0,C 180,E1 -22434.644,E2 -22434.644} C_VEL
LIN {X 0,Y 187.576,Z 440.199,A -85,B 0,C 180,E1 -22436.719,E2 -22436.719} C_VEL
LIN {X 0,Y 190.11,Z 433.275,A -85,B 0,C 180,E1 -22438.723,E2 -22438.723} C_VEL
LIN {X 0,Y 192.893,Z 425.101,A -85,B 0,C 180,E1 -22440.669,E2 -22440.669} C_VEL
LIN {X 0,Y 195.54,Z 416.594,A -85,B 0,C 180,E1 -22442.319,E2 -22442.319} C_VEL
LIN {X 0,Y 197.879,Z 407.881,A -85,B 0,C 180,E1 -22443.707,E2 -22443.707} C_VEL
LIN {X 0,Y 200.238,Z 398.129,A -85,B 0,C 180,E1 -22444.927,E2 -22444.927} C_VEL
LIN {X 0,Y 202.208,Z 388.051,A -85,B 0,C 180,E1 -22445.91,E2 -22445.91} C_VEL
LIN {X 0,Y 203.699,Z 378.349,A -85,B 0,C 180,E1 -22446.617,E2 -22446.617} C_VEL
LIN {X 0,Y 204.806,Z 368.036,A -85,B 0,C 180,E1 -22447.149,E2 -22447.149} C_VEL
LIN {X 0,Y 207.057,Z 325.635,A -85,B 0,C 180,E1 -22448.569,E2 -22448.569} C_VEL
LIN {X 0,Y 204.948,Z 312.176,A -85,B 0,C 180,E1 -22449.634,E2 -22449.634} C_VEL
LIN {X 0,Y 199.785,Z 299.56,A -85,B 0,C 180,E1 -22451.451,E2 -22451.451} C_VEL
LIN {X 0,Y 193.859,Z 287.129,A -85,B 0,C 180,E1 -22453.624,E2 -22453.624} C_VEL
LIN {X 0,Y 187.31,Z 275.341,A -85,B 0,C 180,E1 -22456.185,E2 -22456.185} C_VEL
LIN {X 0,Y 184.886,Z 271.26,A -85,B 0,C 180,E1 -22457.196,E2 -22457.196} C_VEL
LIN {X 0,Y 181.658,Z 266.136,A -85,B 0,C 180,E1 -22458.597,E2 -22458.597} C_VEL
LIN {X 0,Y 179.2,Z 262.257,A -85,B 0,C 180,E1 -22459.767,E2 -22459.767} C_VEL
LIN {X 0,Y 178.709,Z 261.043,A -85,B 0,C 180,E1 -22460.277,E2 -22460.277} C_VEL
LIN {X 0,Y 178.413,Z 259.796,A -85,B 0,C 180,E1 -22461.55,E2 -22461.55} C_VEL
LIN {X 0,Y 178.487,Z 259.721,A -85,B 0,C 180,E1 -22466.545,E2 -22466.545} C_VEL
LIN {X 0,Y 178.523,Z 259.74,A -85,B 0,C 180,E1 -22470.006,E2 -22470.006} C_VEL
LIN {X 0,Y 178.526,Z 259.716,A -85,B 0,C 180,E1 -22474.882,E2 -22474.882} C_VEL
LIN {X 0,Y 178.623,Z 259.686,A -85,B 0,C 180,E1 -22480.785,E2 -22480.785} C_VEL
LIN {X 0,Y 178.651,Z 259.726,A -85,B 0,C 180,E1 -22486.346,E2 -22486.346} C_VEL
LIN {X 0,Y 178.906,Z 259.646,A -85,B 0,C 180,E1 -22490.958,E2 -22490.958} C_VEL
LIN {X 0,Y 179.15,Z 259.635,A -85,B 0,C 180,E1 -22497.75,E2 -22497.75} C_VEL
LIN {X 0,Y 179.368,Z 259.587,A -85,B 0,C 180,E1 -22499.999,E2 -22499.999} C_VEL
LIN {X 0,Y 178.87,Z 259.702,A -85,B 0,C 180,E1 -22504.506,E2 -22504.506} C_VEL
LIN {X 0,Y 178.914,Z 259.648,A -85,B 0,C 180,E1 -22509.039,E2 -22509.039} C_VEL
LIN {X 0,Y 178.663,Z 259.722,A -85,B 0,C 180,E1 -22513.65,E2 -22513.65} C_VEL
LIN {X 0,Y 178.648,Z 259.687,A -85,B 0,C 180,E1 -22518.343,E2 -22518.343} C_VEL
LIN {X 0,Y 178.497,Z 259.752,A -85,B 0,C 180,E1 -22523.186,E2 -22523.186} C_VEL
LIN {X 0,Y 178.482,Z 259.716,A -85,B 0,C 180,E1 -22528.196,E2 -22528.196} C_VEL
LIN {X 0,Y 178.496,Z 259.751,A -85,B 0,C 180,E1 -22530.786,E2 -22530.786} C_VEL
LIN {X 0,Y 178.482,Z 259.723,A -85,B 0,C 180,E1 -22534.218,E2 -22534.218} C_VEL
LIN {X 0,Y 178.509,Z 259.883,A -85,B 0,C 180,E1 -22539.773,E2 -22539.773} C_VEL
LIN {X 0,Y 178.744,Z 260.848,A -85,B 0,C 180,E1 -22540.354,E2 -22540.354} C_VEL
LIN {X 0,Y 180.363,Z 263.689,A -85,B 0,C 180,E1 -22541.174,E2 -22541.174} C_VEL
LIN {X 0,Y 182.001,Z 265.319,A -85,B 0,C 180,E1 -22541.859,E2 -22541.859} C_VEL
LIN {X 0,Y 184.067,Z 268.52,A -85,B 0,C 180,E1 -22542.757,E2 -22542.757} C_VEL
LIN {X 0,Y 185.442,Z 270.304,A -85,B 0,C 180,E1 -22543.317,E2 -22543.317} C_VEL
LIN {X 0,Y 193.246,Z 281.924,A -85,B 0,C 180,E1 -22546.323,E2 -22546.323} C_VEL
LIN {X 0,Y 200.142,Z 293.438,A -85,B 0,C 180,E1 -22548.734,E2 -22548.734} C_VEL
LIN {X 0,Y 207.398,Z 307.661,A -85,B 0,C 180,E1 -22551.106,E2 -22551.106} C_VEL
LIN {X 0,Y 216.251,Z 326.345,A -85,B 0,C 180,E1 -22553.746,E2 -22553.746} C_VEL
LIN {X 0,Y 224.701,Z 340.321,A -85,B 0,C 180,E1 -22555.853,E2 -22555.853} C_VEL
LIN {X 0,Y 233.474,Z 352.37,A -85,B 0,C 180,E1 -22557.742,E2 -22557.742} C_VEL
LIN {X 0,Y 243.637,Z 364.439,A -85,B 0,C 180,E1 -22559.822,E2 -22559.822} C_VEL
LIN {X 0,Y 254.503,Z 376.051,A -85,B 0,C 180,E1 -22562.086,E2 -22562.086} C_VEL
LIN {X 0,Y 266.631,Z 387.191,A -85,B 0,C 180,E1 -22564.524,E2 -22564.524} C_VEL
LIN {X 0,Y 280.005,Z 397.815,A -85,B 0,C 180,E1 -22567.07,E2 -22567.07} C_VEL
LIN {X 0,Y 292.767,Z 407.199,A -85,B 0,C 180,E1 -22569.422,E2 -22569.422} C_VEL
LIN {X 0,Y 300.114,Z 412.668,A -85,B 0,C 180,E1 -22570.862,E2 -22570.862} C_VEL
LIN {X 0,Y 307.409,Z 417.781,A -85,B 0,C 180,E1 -22572.425,E2 -22572.425} C_VEL
LIN {X 0,Y 314.203,Z 422.599,A -85,B 0,C 180,E1 -22574.111,E2 -22574.111} C_VEL
LIN {X 0,Y 321.082,Z 427.22,A -85,B 0,C 180,E1 -22576.068,E2 -22576.068} C_VEL
LIN {X 0,Y 325.82,Z 430.063,A -85,B 0,C 180,E1 -22577.543,E2 -22577.543} C_VEL
LIN {X 0,Y 331.105,Z 433.861,A -85,B 0,C 180,E1 -22579.673,E2 -22579.673} C_VEL
LIN {X 0,Y 335.089,Z 436.385,A -85,B 0,C 180,E1 -22581.558,E2 -22581.558} C_VEL
LIN {X 0,Y 337.435,Z 437.671,A -85,B 0,C 180,E1 -22582.821,E2 -22582.821} C_VEL
LIN {X 0,Y 339.448,Z 438.647,A -85,B 0,C 180,E1 -22584.058,E2 -22584.058} C_VEL
LIN {X 0,Y 341.108,Z 439.386,A -85,B 0,C 180,E1 -22585.273,E2 -22585.273} C_VEL
LIN {X 0,Y 342.472,Z 439.856,A -85,B 0,C 180,E1 -22586.47,E2 -22586.47} C_VEL
LIN {X 0,Y 343.327,Z 440.236,A -85,B 0,C 180,E1 -22587.654,E2 -22587.654} C_VEL
LIN {X 0,Y 343.774,Z 440.503,A -85,B 0,C 180,E1 -22588.829,E2 -22588.829} C_VEL
LIN {X 0,Y 344.062,Z 440.474,A -85,B 0,C 180,E1 -22590,E2 -22590} C_VEL
LIN {X 0,Y 343.794,Z 440.473,A -85,B 0,C 180,E1 -22591.171,E2 -22591.171} C_VEL
LIN {X 0,Y 343.351,Z 440.193,A -85,B 0,C 180,E1 -22592.346,E2 -22592.346} C_VEL
LIN {X 0,Y 342.447,Z 439.844,A -85,B 0,C 180,E1 -22593.53,E2 -22593.53} C_VEL
LIN {X 0,Y 341.087,Z 439.365,A -85,B 0,C 180,E1 -22594.728,E2 -22594.728} C_VEL
LIN {X 0,Y 339.233,Z 438.56,A -85,B 0,C 180,E1 -22596.056,E2 -22596.056} C_VEL
LIN {X 0,Y 337.422,Z 437.655,A -85,B 0,C 180,E1 -22597.179,E2 -22597.179} C_VEL
LIN {X 0,Y 334.285,Z 435.923,A -85,B 0,C 180,E1 -22598.843,E2 -22598.843} C_VEL
LIN {X 0,Y 331.127,Z 433.842,A -85,B 0,C 180,E1 -22600.326,E2 -22600.326} C_VEL
LIN {X 0,Y 325.812,Z 430.057,A -85,B 0,C 180,E1 -22602.457,E2 -22602.457} C_VEL
LIN {X 0,Y 319.321,Z 426.119,A -85,B 0,C 180,E1 -22604.444,E2 -22604.444} C_VEL
LIN {X 0,Y 314.201,Z 422.609,A -85,B 0,C 180,E1 -22605.887,E2 -22605.887} C_VEL
LIN {X 0,Y 307.417,Z 417.769,A -85,B 0,C 180,E1 -22607.58,E2 -22607.58} C_VEL
LIN {X 0,Y 300.157,Z 412.692,A -85,B 0,C 180,E1 -22609.135,E2 -22609.135} C_VEL
LIN {X 0,Y 292.76,Z 407.228,A -85,B 0,C 180,E1 -22610.574,E2 -22610.574} C_VEL
LIN {X 0,Y 278.098,Z 396.352,A -85,B 0,C 180,E1 -22613.29,E2 -22613.29} C_VEL
LIN {X 0,Y 265.282,Z 385.999,A -85,B 0,C 180,E1 -22615.746,E2 -22615.746} C_VEL
LIN {X 0,Y 253.577,Z 375.119,A -85,B 0,C 180,E1 -22618.11,E2 -22618.11} C_VEL
LIN {X 0,Y 242.465,Z 363.067,A -85,B 0,C 180,E1 -22620.424,E2 -22620.424} C_VEL
LIN {X 0,Y 232.753,Z 351.522,A -85,B 0,C 180,E1 -22622.401,E2 -22622.401} C_VEL
LIN {X 0,Y 222.723,Z 337.345,A -85,B 0,C 180,E1 -22624.61,E2 -22624.61} C_VEL
LIN {X 0,Y 215.036,Z 324.025,A -85,B 0,C 180,E1 -22626.588,E2 -22626.588} C_VEL
LIN {X 0,Y 205.23,Z 303.245,A -85,B 0,C 180,E1 -22629.584,E2 -22629.584} C_VEL
LIN {X 0,Y 198.278,Z 290.182,A -85,B 0,C 180,E1 -22631.899,E2 -22631.899} C_VEL
LIN {X 0,Y 191.604,Z 279.45,A -85,B 0,C 180,E1 -22634.278,E2 -22634.278} C_VEL
LIN {X 0,Y 187.038,Z 272.739,A -85,B 0,C 180,E1 -22636.031,E2 -22636.031} C_VEL
LIN {X 0,Y 184.471,Z 268.993,A -85,B 0,C 180,E1 -22637.08,E2 -22637.08} C_VEL
LIN {X 0,Y 182.371,Z 266.077,A -85,B 0,C 180,E1 -22637.967,E2 -22637.967} C_VEL
LIN {X 0,Y 181.611,Z 264.798,A -85,B 0,C 180,E1 -22638.31,E2 -22638.31} C_VEL
LIN {X 0,Y 179.489,Z 262.536,A -85,B 0,C 180,E1 -22639.218,E2 -22639.218} C_VEL
LIN {X 0,Y 178.585,Z 260.28,A -85,B 0,C 180,E1 -22639.88,E2 -22639.88} C_VEL
LIN {X 0,Y 178.476,Z 259.779,A -85,B 0,C 180,E1 -22640.584,E2 -22640.584} C_VEL
LIN {X 0,Y 178.482,Z 259.723,A -85,B 0,C 180,E1 -22645.782,E2 -22645.782} C_VEL
LIN {X 0,Y 178.519,Z 259.733,A -85,B 0,C 180,E1 -22650.008,E2 -22650.008} C_VEL
LIN {X 0,Y 178.518,Z 259.726,A -85,B 0,C 180,E1 -22654.887,E2 -22654.887} C_VEL
LIN {X 0,Y 178.62,Z 259.688,A -85,B 0,C 180,E1 -22660.787,E2 -22660.787} C_VEL
LIN {X 0,Y 178.661,Z 259.716,A -85,B 0,C 180,E1 -22664.018,E2 -22664.018} C_VEL
LIN {X 0,Y 178.834,Z 259.658,A -85,B 0,C 180,E1 -22669.257,E2 -22669.257} C_VEL
LIN {X 0,Y 178.915,Z 259.679,A -85,B 0,C 180,E1 -22673.234,E2 -22673.234} C_VEL
LIN {X 0,Y 179.153,Z 259.627,A -85,B 0,C 180,E1 -22677.753,E2 -22677.753} C_VEL
LIN {X 0,Y 179.368,Z 259.587,A -85,B 0,C 180,E1 -22680.001,E2 -22680.001} C_VEL
LIN {X 0,Y 178.862,Z 259.705,A -85,B 0,C 180,E1 -22684.509,E2 -22684.509} C_VEL
LIN {X 0,Y 178.906,Z 259.646,A -85,B 0,C 180,E1 -22689.042,E2 -22689.042} C_VEL
LIN {X 0,Y 178.651,Z 259.726,A -85,B 0,C 180,E1 -22693.654,E2 -22693.654} C_VEL
LIN {X 0,Y 178.623,Z 259.686,A -85,B 0,C 180,E1 -22699.215,E2 -22699.215} C_VEL
LIN {X 0,Y 178.526,Z 259.716,A -85,B 0,C 180,E1 -22705.118,E2 -22705.118} C_VEL
LIN {X 0,Y 178.501,Z 259.751,A -85,B 0,C 180,E1 -22710.788,E2 -22710.788} C_VEL
LIN {X 0,Y 178.486,Z 259.72,A -85,B 0,C 180,E1 -22714.22,E2 -22714.22} C_VEL
LIN {X 0,Y 178.426,Z 259.968,A -85,B 0,C 180,E1 -22718.757,E2 -22718.757} C_VEL
LIN {X 0,Y 178.932,Z 261.603,A -85,B 0,C 180,E1 -22720.03,E2 -22720.03} C_VEL
LIN {X 0,Y 181.266,Z 265.645,A -85,B 0,C 180,E1 -22721.234,E2 -22721.234} C_VEL
LIN {X 0,Y 182.942,Z 268.117,A -85,B 0,C 180,E1 -22721.967,E2 -22721.967} C_VEL
LIN {X 0,Y 186.337,Z 273.694,A -85,B 0,C 180,E1 -22723.414,E2 -22723.414} C_VEL
LIN {X 0,Y 191.755,Z 283.273,A -85,B 0,C 180,E1 -22725.581,E2 -22725.581} C_VEL
LIN {X 0,Y 196.9,Z 293.188,A -85,B 0,C 180,E1 -22727.501,E2 -22727.501} C_VEL
LIN {X 0,Y 203.171,Z 307.606,A -85,B 0,C 180,E1 -22729.747,E2 -22729.747} C_VEL
LIN {X 0,Y 205.2,Z 313.069,A -85,B 0,C 180,E1 -22730.464,E2 -22730.464} C_VEL
LIN {X 0,Y 207.022,Z 326.092,A -85,B 0,C 180,E1 -22731.443,E2 -22731.443} C_VEL
LIN {X 0,Y 204.789,Z 368.14,A -85,B 0,C 180,E1 -22732.848,E2 -22732.848} C_VEL
LIN {X 0,Y 203.636,Z 378.969,A -85,B 0,C 180,E1 -22733.424,E2 -22733.424} C_VEL
LIN {X 0,Y 201.985,Z 389.338,A -85,B 0,C 180,E1 -22734.198,E2 -22734.198} C_VEL
LIN {X 0,Y 199.581,Z 401.148,A -85,B 0,C 180,E1 -22735.402,E2 -22735.402} C_VEL
LIN {X 0,Y 196.701,Z 412.541,A -85,B 0,C 180,E1 -22736.984,E2 -22736.984} C_VEL
LIN {X 0,Y 193.658,Z 422.834,A -85,B 0,C 180,E1 -22738.859,E2 -22738.859} C_VEL
LIN {X 0,Y 190.808,Z 431.358,A -85,B 0,C 180,E1 -22740.789,E2 -22740.789} C_VEL
LIN {X 0,Y 188.177,Z 438.573,A -85,B 0,C 180,E1 -22742.774,E2 -22742.774} C_VEL
LIN {X 0,Y 185.902,Z 444.774,A -85,B 0,C 180,E1 -22744.83,E2 -22744.83} C_VEL
LIN {X 0,Y 183.454,Z 451.314,A -85,B 0,C 180,E1 -22747.475,E2 -22747.475} C_VEL
LIN {X 0,Y 181.597,Z 455.813,A -85,B 0,C 180,E1 -22749.616,E2 -22749.616} C_VEL
LIN {X 0,Y 179.367,Z 461.305,A -85,B 0,C 180,E1 -22752.91,E2 -22752.91} C_VEL
LIN {X 0,Y 177.766,Z 465.634,A -85,B 0,C 180,E1 -22756.278,E2 -22756.278} C_VEL
LIN {X 0,Y 176.979,Z 468.03,A -85,B 0,C 180,E1 -22758.579,E2 -22758.579} C_VEL
LIN {X 0,Y 176.46,Z 469.809,A -85,B 0,C 180,E1 -22760.833,E2 -22760.833} C_VEL
LIN {X 0,Y 176.01,Z 472.267,A -85,B 0,C 180,E1 -22765.42,E2 -22765.42} C_VEL
LIN {X 0,Y 175.968,Z 472.907,A -85,B 0,C 180,E1 -22768.385,E2 -22768.385} C_VEL
LIN {X 0,Y 175.294,Z 473.015,A -85,B 0,C 180,E1 -22770.295,E2 -22770.295} C_VEL
LIN {X 0,Y 173.682,Z 472.835,A -85,B 0,C 180,E1 -22772.173,E2 -22772.173} C_VEL
LIN {X 0,Y 170.032,Z 471.613,A -85,B 0,C 180,E1 -22775.971,E2 -22775.971} C_VEL
LIN {X 0,Y 169.174,Z 470.453,A -85,B 0,C 180,E1 -22778.277,E2 -22778.277} C_VEL
LIN {X 0,Y 169.207,Z 470.166,A -85,B 0,C 180,E1 -22778.609,E2 -22778.609} C_VEL
LIN {X 0,Y 170.015,Z 467.812,A -85,B 0,C 180,E1 -22781.928,E2 -22781.928} C_VEL
LIN {X 0,Y 171.298,Z 464.197,A -85,B 0,C 180,E1 -22785.467,E2 -22785.467} C_VEL
LIN {X 0,Y 173.313,Z 459.452,A -85,B 0,C 180,E1 -22788.93,E2 -22788.93} C_VEL
LIN {X 0,Y 175.876,Z 453.43,A -85,B 0,C 180,E1 -22792.31,E2 -22792.31} C_VEL
LIN {X 0,Y 178.302,Z 447.574,A -85,B 0,C 180,E1 -22794.961,E2 -22794.961} C_VEL
LIN {X 0,Y 180.638,Z 441.633,A -85,B 0,C 180,E1 -22797.203,E2 -22797.203} C_VEL
LIN {X 0,Y 183.91,Z 433.082,A -85,B 0,C 180,E1 -22799.788,E2 -22799.788} C_VEL
LIN {X 0,Y 186.807,Z 424.908,A -85,B 0,C 180,E1 -22801.783,E2 -22801.783} C_VEL
LIN {X 0,Y 189.572,Z 416.401,A -85,B 0,C 180,E1 -22803.467,E2 -22803.467} C_VEL
LIN {X 0,Y 192.007,Z 407.688,A -85,B 0,C 180,E1 -22804.884,E2 -22804.884} C_VEL
LIN {X 0,Y 194.461,Z 397.936,A -85,B 0,C 180,E1 -22806.125,E2 -22806.125} C_VEL
LIN {X 0,Y 196.514,Z 387.859,A -85,B 0,C 180,E1 -22807.121,E2 -22807.121} C_VEL
LIN {X 0,Y 198.068,Z 378.022,A -85,B 0,C 180,E1 -22807.85,E2 -22807.85} C_VEL
LIN {X 0,Y 199.157,Z 368.377,A -85,B 0,C 180,E1 -22808.358,E2 -22808.358} C_VEL
LIN {X 0,Y 200.889,Z 338.166,A -85,B 0,C 180,E1 -22809.408,E2 -22809.408} C_VEL
LIN {X 0,Y 201.389,Z 325.884,A -85,B 0,C 180,E1 -22809.847,E2 -22809.847} C_VEL
LIN {X 0,Y 199.701,Z 314.961,A -85,B 0,C 180,E1 -22810.754,E2 -22810.754} C_VEL
LIN {X 0,Y 193.738,Z 300.469,A -85,B 0,C 180,E1 -22812.994,E2 -22812.994} C_VEL
LIN {X 0,Y 188.866,Z 290.275,A -85,B 0,C 180,E1 -22814.91,E2 -22814.91} C_VEL
LIN {X 0,Y 181.511,Z 276.927,A -85,B 0,C 180,E1 -22818.023,E2 -22818.023} C_VEL
LIN {X 0,Y 177.741,Z 271.002,A -85,B 0,C 180,E1 -22819.743,E2 -22819.743} C_VEL
LIN {X 0,Y 174.679,Z 266.258,A -85,B 0,C 180,E1 -22821.238,E2 -22821.238} C_VEL
LIN {X 0,Y 172.037,Z 262.824,A -85,B 0,C 180,E1 -22822.577,E2 -22822.577} C_VEL
LIN {X 0,Y 171.464,Z 261.176,A -85,B 0,C 180,E1 -22823.168,E2 -22823.168} C_VEL
LIN {X 0,Y 171.405,Z 260.676,A -85,B 0,C 180,E1 -22823.883,E2 -22823.883} C_VEL
LIN {X 0,Y 171.458,Z 260.628,A -85,B 0,C 180,E1 -22829.404,E2 -22829.404} C_VEL
LIN {X 0,Y 171.463,Z 260.59,A -85,B 0,C 180,E1 -22834.388,E2 -22834.388} C_VEL
LIN {X 0,Y 171.578,Z 260.562,A -85,B 0,C 180,E1 -22840.87,E2 -22840.87} C_VEL
LIN {X 0,Y 171.569,Z 260.611,A -85,B 0,C 180,E1 -22845.771,E2 -22845.771} C_VEL
LIN {X 0,Y 171.844,Z 260.524,A -85,B 0,C 180,E1 -22850.583,E2 -22850.583} C_VEL
LIN {X 0,Y 171.81,Z 260.584,A -85,B 0,C 180,E1 -22855.306,E2 -22855.306} C_VEL
LIN {X 0,Y 172.331,Z 260.463,A -85,B 0,C 180,E1 -22859.999,E2 -22859.999} C_VEL
LIN {X 0,Y 171.819,Z 260.581,A -85,B 0,C 180,E1 -22864.691,E2 -22864.691} C_VEL
LIN {X 0,Y 171.85,Z 260.526,A -85,B 0,C 180,E1 -22869.414,E2 -22869.414} C_VEL
LIN {X 0,Y 171.591,Z 260.61,A -85,B 0,C 180,E1 -22874.225,E2 -22874.225} C_VEL
LIN {X 0,Y 171.539,Z 260.57,A -85,B 0,C 180,E1 -22879.556,E2 -22879.556} C_VEL
LIN {X 0,Y 171.456,Z 260.598,A -85,B 0,C 180,E1 -22885.607,E2 -22885.607} C_VEL
LIN {X 0,Y 171.454,Z 260.623,A -85,B 0,C 180,E1 -22890.594,E2 -22890.594} C_VEL
